LIN {X 0,Y 587.637,Z 719.821,A -85,B 0,C 180,E1 26964.756,E2 26964.756} C_VEL
LIN {X 0,Y 588.575,Z 722.928,A -85,B 0,C 180,E1 26962.657,E2 26962.657} C_VEL
LIN {X 0,Y 589.247,Z 724.472,A -85,B 0,C 180,E1 26961.936,E2 26961.936} C_VEL
LIN {X 0,Y 590.735,Z 728.438,A -85,B 0,C 180,E1 26960.6,E2 26960.6} C_VEL
LIN {X 0,Y 592.603,Z 733.926,A -85,B 0,C 180,E1 26959.233,E2 26959.233} C_VEL
LIN {X 0,Y 593.872,Z 738.208,A -85,B 0,C 180,E1 26958.376,E2 26958.376} C_VEL
LIN {X 0,Y 585.951,Z 770.314,A -85,B 0,C 180,E1 26955.875,E2 26955.875} C_VEL
LIN {X 0,Y 580.418,Z 801.749,A -85,B 0,C 180,E1 26953.509,E2 26953.509} C_VEL
LIN {X 0,Y 578.896,Z 823.206,A -85,B 0,C 180,E1 26951.811,E2 26951.811} C_VEL
LIN {X 0,Y 579.57,Z 841.188,A -85,B 0,C 180,E1 26950.31,E2 26950.31} C_VEL
LIN {X 0,Y 582.431,Z 858.387,A -85,B 0,C 180,E1 26948.793,E2 26948.793} C_VEL
LIN {X 0,Y 587.132,Z 873.472,A -85,B 0,C 180,E1 26947.396,E2 26947.396} C_VEL
LIN {X 0,Y 593.648,Z 887.403,A -85,B 0,C 180,E1 26946.053,E2 26946.053} C_VEL
LIN {X 0,Y 602.264,Z 900.569,A -85,B 0,C 180,E1 26944.733,E2 26944.733} C_VEL
LIN {X 0,Y 611.989,Z 911.844,A -85,B 0,C 180,E1 26943.565,E2 26943.565} C_VEL
LIN {X 0,Y 613.681,Z 913.685,A -85,B 0,C 180,E1 26943.378,E2 26943.378} C_VEL
LIN {X 0,Y 600.72,Z 934.889,A -85,B 0,C 180,E1 26942.747,E2 26942.747} C_VEL
LIN {X 0,Y 591.048,Z 953.679,A -85,B 0,C 180,E1 26942.084,E2 26942.084} C_VEL
LIN {X 0,Y 583.725,Z 969.894,A -85,B 0,C 180,E1 26941.455,E2 26941.455} C_VEL
LIN {X 0,Y 576.421,Z 987.193,A -85,B 0,C 180,E1 26940.746,E2 26940.746} C_VEL
LIN {X 0,Y 572.039,Z 1000.302,A -85,B 0,C 180,E1 26940.18,E2 26940.18} C_VEL
LIN {X 0,Y 569.588,Z 1022.689,A -85,B 0,C 180,E1 26939.955,E2 26939.955} C_VEL
LIN {X 0,Y 568.415,Z 1062.738,A -85,B 0,C 180,E1 26939.349,E2 26939.349} C_VEL
LIN {X 0,Y 567.38,Z 1084.854,A -85,B 0,C 180,E1 26938.837,E2 26938.837} C_VEL
LIN {X 0,Y 566.128,Z 1105.829,A -85,B 0,C 180,E1 26938.174,E2 26938.174} C_VEL
LIN {X 0,Y 564.559,Z 1128.324,A -85,B 0,C 180,E1 26937.264,E2 26937.264} C_VEL
LIN {X 0,Y 562.987,Z 1148.678,A -85,B 0,C 180,E1 26936.245,E2 26936.245} C_VEL
LIN {X 0,Y 561.314,Z 1168.753,A -85,B 0,C 180,E1 26935.026,E2 26935.026} C_VEL
LIN {X 0,Y 559.661,Z 1187.098,A -85,B 0,C 180,E1 26933.7,E2 26933.7} C_VEL
LIN {X 0,Y 558.095,Z 1204.72,A -85,B 0,C 180,E1 26932.21,E2 26932.21} C_VEL
LIN {X 0,Y 556.649,Z 1220.957,A -85,B 0,C 180,E1 26930.612,E2 26930.612} C_VEL
LIN {X 0,Y 555.379,Z 1235.689,A -85,B 0,C 180,E1 26928.907,E2 26928.907} C_VEL
LIN {X 0,Y 554.298,Z 1249.482,A -85,B 0,C 180,E1 26927.047,E2 26927.047} C_VEL
LIN {X 0,Y 553.424,Z 1261.927,A -85,B 0,C 180,E1 26925.078,E2 26925.078} C_VEL
LIN {X 0,Y 552.819,Z 1272.613,A -85,B 0,C 180,E1 26923.065,E2 26923.065} C_VEL
LIN {X 0,Y 552.412,Z 1281.385,A -85,B 0,C 180,E1 26921.06,E2 26921.06} C_VEL
LIN {X 0,Y 552.19,Z 1288.893,A -85,B 0,C 180,E1 26918.957,E2 26918.957} C_VEL
LIN {X 0,Y 552.095,Z 1294.66,A -85,B 0,C 180,E1 26916.864,E2 26916.864} C_VEL
LIN {X 0,Y 552.078,Z 1298.97,A -85,B 0,C 180,E1 26914.673,E2 26914.673} C_VEL
LIN {X 0,Y 552.098,Z 1301.66,A -85,B 0,C 180,E1 26912.49,E2 26912.49} C_VEL
LIN {X 0,Y 552.111,Z 1302.611,A -85,B 0,C 180,E1 26910.414,E2 26910.414} C_VEL
LIN {X 0,Y 552.119,Z 1302.041,A -85,B 0,C 180,E1 26908.234,E2 26908.234} C_VEL
LIN {X 0,Y 552.092,Z 1299.995,A -85,B 0,C 180,E1 26906.156,E2 26906.156} C_VEL
LIN {X 0,Y 552.096,Z 1296.342,A -85,B 0,C 180,E1 26904.073,E2 26904.073} C_VEL
LIN {X 0,Y 552.146,Z 1291.188,A -85,B 0,C 180,E1 26901.983,E2 26901.983} C_VEL
LIN {X 0,Y 552.298,Z 1284.244,A -85,B 0,C 180,E1 26899.885,E2 26899.885} C_VEL
LIN {X 0,Y 552.609,Z 1275.501,A -85,B 0,C 180,E1 26897.777,E2 26897.777} C_VEL
LIN {X 0,Y 553.09,Z 1265.374,A -85,B 0,C 180,E1 26895.766,E2 26895.766} C_VEL
LIN {X 0,Y 553.776,Z 1253.837,A -85,B 0,C 180,E1 26893.854,E2 26893.854} C_VEL
LIN {X 0,Y 554.714,Z 1240.173,A -85,B 0,C 180,E1 26891.937,E2 26891.937} C_VEL
LIN {X 0,Y 555.856,Z 1225.016,A -85,B 0,C 180,E1 26890.123,E2 26890.123} C_VEL
LIN {X 0,Y 557.166,Z 1208.907,A -85,B 0,C 180,E1 26888.47,E2 26888.47} C_VEL
LIN {X 0,Y 558.616,Z 1191.119,A -85,B 0,C 180,E1 26886.92,E2 26886.92} C_VEL
LIN {X 0,Y 560.211,Z 1171.724,A -85,B 0,C 180,E1 26885.481,E2 26885.481} C_VEL
LIN {X 0,Y 561.815,Z 1151.511,A -85,B 0,C 180,E1 26884.21,E2 26884.21} C_VEL
LIN {X 0,Y 563.458,Z 1130.214,A -85,B 0,C 180,E1 26883.094,E2 26883.094} C_VEL
LIN {X 0,Y 565.016,Z 1107.978,A -85,B 0,C 180,E1 26882.147,E2 26882.147} C_VEL
LIN {X 0,Y 566.431,Z 1085.264,A -85,B 0,C 180,E1 26881.387,E2 26881.387} C_VEL
LIN {X 0,Y 567.595,Z 1062.247,A -85,B 0,C 180,E1 26880.821,E2 26880.821} C_VEL
LIN {X 0,Y 568.909,Z 1024.211,A -85,B 0,C 180,E1 26880.177,E2 26880.177} C_VEL
LIN {X 0,Y 570.051,Z 1012.277,A -85,B 0,C 180,E1 26880.006,E2 26880.006} C_VEL
LIN {X 0,Y 578.286,Z 988.02,A -85,B 0,C 180,E1 26878.869,E2 26878.869} C_VEL
LIN {X 0,Y 585.721,Z 971.102,A -85,B 0,C 180,E1 26878.163,E2 26878.163} C_VEL
LIN {X 0,Y 597.338,Z 946.651,A -85,B 0,C 180,E1 26877.213,E2 26877.213} C_VEL
LIN {X 0,Y 608.71,Z 926.849,A -85,B 0,C 180,E1 26876.56,E2 26876.56} C_VEL
LIN {X 0,Y 615.537,Z 915.878,A -85,B 0,C 180,E1 26876.237,E2 26876.237} C_VEL
LIN {X 0,Y 605.204,Z 904.179,A -85,B 0,C 180,E1 26875.032,E2 26875.032} C_VEL
LIN {X 0,Y 596.035,Z 890.457,A -85,B 0,C 180,E1 26873.714,E2 26873.714} C_VEL
LIN {X 0,Y 588.846,Z 875.63,A -85,B 0,C 180,E1 26872.386,E2 26872.386} C_VEL
LIN {X 0,Y 583.433,Z 859.428,A -85,B 0,C 180,E1 26871.025,E2 26871.025} C_VEL
LIN {X 0,Y 579.733,Z 840.872,A -85,B 0,C 180,E1 26869.57,E2 26869.57} C_VEL
LIN {X 0,Y 578.123,Z 820.933,A -85,B 0,C 180,E1 26868.117,E2 26868.117} C_VEL
LIN {X 0,Y 578.452,Z 797.639,A -85,B 0,C 180,E1 26866.53,E2 26866.53} C_VEL
LIN {X 0,Y 583.409,Z 741.175,A -85,B 0,C 180,E1 26862.876,E2 26862.876} C_VEL
LIN {X 0,Y 584.291,Z 731.836,A -85,B 0,C 180,E1 26862.263,E2 26862.263} C_VEL
LIN {X 0,Y 572.986,Z 706.025,A -85,B 0,C 180,E1 26859.37,E2 26859.37} C_VEL
LIN {X 0,Y 570.213,Z 699.791,A -85,B 0,C 180,E1 26858.62,E2 26858.62} C_VEL
LIN {X 0,Y 572.694,Z 699.884,A -85,B 0,C 180,E1 26858.135,E2 26858.135} C_VEL
LIN {X 0,Y 575.711,Z 710.211,A -85,B 0,C 180,E1 26856.44,E2 26856.44} C_VEL
LIN {X 0,Y 576.967,Z 715.049,A -85,B 0,C 180,E1 26855.777,E2 26855.777} C_VEL
LIN {X 0,Y 580.175,Z 722.589,A -85,B 0,C 180,E1 26855.137,E2 26855.137} C_VEL
LIN {X 0,Y 582.997,Z 739.875,A -85,B 0,C 180,E1 26854.313,E2 26854.313} C_VEL
LIN {X 0,Y 576.786,Z 834.739,A -85,B 0,C 180,E1 26852.485,E2 26852.485} C_VEL
LIN {X 0,Y 572.384,Z 927.388,A -85,B 0,C 180,E1 26850.83,E2 26850.83} C_VEL
LIN {X 0,Y 569.328,Z 1016.488,A -85,B 0,C 180,E1 26849.344,E2 26849.344} C_VEL
LIN {X 0,Y 568.303,Z 1039.379,A -85,B 0,C 180,E1 26848.764,E2 26848.764} C_VEL
LIN {X 0,Y 567.075,Z 1060.726,A -85,B 0,C 180,E1 26848.046,E2 26848.046} C_VEL
LIN {X 0,Y 565.582,Z 1082.832,A -85,B 0,C 180,E1 26847.104,E2 26847.104} C_VEL
LIN {X 0,Y 564.08,Z 1102.487,A -85,B 0,C 180,E1 26846.079,E2 26846.079} C_VEL
LIN {X 0,Y 562.432,Z 1121.912,A -85,B 0,C 180,E1 26844.863,E2 26844.863} C_VEL
LIN {X 0,Y 560.743,Z 1140.326,A -85,B 0,C 180,E1 26843.487,E2 26843.487} C_VEL
LIN {X 0,Y 559.062,Z 1157.806,A -85,B 0,C 180,E1 26841.95,E2 26841.95} C_VEL
LIN {X 0,Y 557.574,Z 1173.309,A -85,B 0,C 180,E1 26840.359,E2 26840.359} C_VEL
LIN {X 0,Y 556.152,Z 1188.302,A -85,B 0,C 180,E1 26838.556,E2 26838.556} C_VEL
LIN {X 0,Y 554.91,Z 1201.645,A -85,B 0,C 180,E1 26836.649,E2 26836.649} C_VEL
LIN {X 0,Y 553.906,Z 1213.516,A -85,B 0,C 180,E1 26834.639,E2 26834.639} C_VEL
LIN {X 0,Y 553.135,Z 1223.889,A -85,B 0,C 180,E1 26832.528,E2 26832.528} C_VEL
LIN {X 0,Y 552.629,Z 1232.359,A -85,B 0,C 180,E1 26830.424,E2 26830.424} C_VEL
LIN {X 0,Y 552.285,Z 1239.262,A -85,B 0,C 180,E1 26828.223,E2 26828.223} C_VEL
LIN {X 0,Y 552.102,Z 1244.436,A -85,B 0,C 180,E1 26826.03,E2 26826.03} C_VEL
LIN {X 0,Y 552.013,Z 1248.008,A -85,B 0,C 180,E1 26823.843,E2 26823.843} C_VEL
LIN {X 0,Y 551.984,Z 1249.897,A -85,B 0,C 180,E1 26821.661,E2 26821.661} C_VEL
LIN {X 0,Y 551.985,Z 1250.235,A -85,B 0,C 180,E1 26819.377,E2 26819.377} C_VEL
LIN {X 0,Y 551.983,Z 1248.966,A -85,B 0,C 180,E1 26817.136,E2 26817.136} C_VEL
LIN {X 0,Y 552.025,Z 1246.172,A -85,B 0,C 180,E1 26815.012,E2 26815.012} C_VEL
LIN {X 0,Y 552.147,Z 1241.721,A -85,B 0,C 180,E1 26812.822,E2 26812.822} C_VEL
LIN {X 0,Y 552.383,Z 1235.625,A -85,B 0,C 180,E1 26810.624,E2 26810.624} C_VEL
LIN {X 0,Y 552.774,Z 1228.041,A -85,B 0,C 180,E1 26808.523,E2 26808.523} C_VEL
LIN {X 0,Y 553.376,Z 1218.633,A -85,B 0,C 180,E1 26806.414,E2 26806.414} C_VEL
LIN {X 0,Y 554.213,Z 1207.87,A -85,B 0,C 180,E1 26804.406,E2 26804.406} C_VEL
LIN {X 0,Y 555.271,Z 1195.735,A -85,B 0,C 180,E1 26802.499,E2 26802.499} C_VEL
LIN {X 0,Y 556.51,Z 1182.18,A -85,B 0,C 180,E1 26800.695,E2 26800.695} C_VEL
LIN {X 0,Y 558.041,Z 1166.325,A -85,B 0,C 180,E1 26798.891,E2 26798.891} C_VEL
LIN {X 0,Y 559.663,Z 1149.96,A -85,B 0,C 180,E1 26797.3,E2 26797.3} C_VEL
LIN {X 0,Y 561.374,Z 1132.001,A -85,B 0,C 180,E1 26795.816,E2 26795.816} C_VEL
LIN {X 0,Y 563.033,Z 1113.854,A -85,B 0,C 180,E1 26794.547,E2 26794.547} C_VEL
LIN {X 0,Y 564.757,Z 1093.28,A -85,B 0,C 180,E1 26793.332,E2 26793.332} C_VEL
LIN {X 0,Y 566.359,Z 1072.777,A -85,B 0,C 180,E1 26792.334,E2 26792.334} C_VEL
LIN {X 0,Y 567.755,Z 1051.302,A -85,B 0,C 180,E1 26791.493,E2 26791.493} C_VEL
LIN {X 0,Y 568.91,Z 1029.578,A -85,B 0,C 180,E1 26790.838,E2 26790.838} C_VEL
LIN {X 0,Y 569.869,Z 1006.211,A -85,B 0,C 180,E1 26790.329,E2 26790.329} C_VEL
LIN {X 0,Y 576.672,Z 748.494,A -85,B 0,C 180,E1 26786.536,E2 26786.536} C_VEL
LIN {X 0,Y 576.781,Z 737.467,A -85,B 0,C 180,E1 26786.358,E2 26786.358} C_VEL
LIN {X 0,Y 571.105,Z 712.252,A -85,B 0,C 180,E1 26785.574,E2 26785.574} C_VEL
LIN {X 0,Y 567.095,Z 704.126,A -85,B 0,C 180,E1 26785.161,E2 26785.161} C_VEL
LIN {X 0,Y 560.021,Z 682.503,A -85,B 0,C 180,E1 26782.611,E2 26782.611} C_VEL
LIN {X 0,Y 553.503,Z 663.719,A -85,B 0,C 180,E1 26780.315,E2 26780.315} C_VEL
LIN {X 0,Y 553.497,Z 663.72,A -85,B 0,C 180,E1 26776.932,E2 26776.932} C_VEL
LIN {X 0,Y 553.509,Z 663.725,A -85,B 0,C 180,E1 26773.494,E2 26773.494} C_VEL
LIN {X 0,Y 553.506,Z 663.721,A -85,B 0,C 180,E1 26770.565,E2 26770.565} C_VEL
LIN {X 0,Y 552.506,Z 663.847,A -85,B 0,C 180,E1 26769.768,E2 26769.768} C_VEL
LIN {X 0,Y 546.084,Z 664.643,A -85,B 0,C 180,E1 26767.529,E2 26767.529} C_VEL
LIN {X 0,Y 545.549,Z 664.706,A -85,B 0,C 180,E1 26766.946,E2 26766.946} C_VEL
LIN {X 0,Y 545.555,Z 664.708,A -85,B 0,C 180,E1 26763.609,E2 26763.609} C_VEL
LIN {X 0,Y 545.566,Z 664.706,A -85,B 0,C 180,E1 26760.11,E2 26760.11} C_VEL
LIN {X 0,Y 545.553,Z 664.71,A -85,B 0,C 180,E1 26756.683,E2 26756.683} C_VEL
LIN {X 0,Y 545.565,Z 664.712,A -85,B 0,C 180,E1 26753.322,E2 26753.322} C_VEL
LIN {X 0,Y 545.567,Z 664.709,A -85,B 0,C 180,E1 26749.821,E2 26749.821} C_VEL
LIN {X 0,Y 545.555,Z 664.713,A -85,B 0,C 180,E1 26746.396,E2 26746.396} C_VEL
LIN {X 0,Y 545.559,Z 664.703,A -85,B 0,C 180,E1 26743.03,E2 26743.03} C_VEL
LIN {X 0,Y 545.552,Z 664.712,A -85,B 0,C 180,E1 26739.709,E2 26739.709} C_VEL
LIN {X 0,Y 545.565,Z 664.709,A -85,B 0,C 180,E1 26736.315,E2 26736.315} C_VEL
LIN {X 0,Y 545.552,Z 664.707,A -85,B 0,C 180,E1 26732.838,E2 26732.838} C_VEL
LIN {X 0,Y 545.548,Z 664.703,A -85,B 0,C 180,E1 26729.476,E2 26729.476} C_VEL
LIN {X 0,Y 545.553,Z 664.702,A -85,B 0,C 180,E1 26726.113,E2 26726.113} C_VEL
LIN {X 0,Y 545.562,Z 664.702,A -85,B 0,C 180,E1 26722.631,E2 26722.631} C_VEL
LIN {X 0,Y 545.549,Z 664.704,A -85,B 0,C 180,E1 26719.227,E2 26719.227} C_VEL
LIN {X 0,Y 545.561,Z 664.706,A -85,B 0,C 180,E1 26715.893,E2 26715.893} C_VEL
LIN {X 0,Y 545.567,Z 664.709,A -85,B 0,C 180,E1 26712.51,E2 26712.51} C_VEL
LIN {X 0,Y 545.561,Z 664.712,A -85,B 0,C 180,E1 26709.062,E2 26709.062} C_VEL
LIN {X 0,Y 545.562,Z 664.713,A -85,B 0,C 180,E1 26705.648,E2 26705.648} C_VEL
LIN {X 0,Y 545.556,Z 664.709,A -85,B 0,C 180,E1 26702.258,E2 26702.258} C_VEL
LIN {X 0,Y 545.565,Z 664.71,A -85,B 0,C 180,E1 26698.86,E2 26698.86} C_VEL
LIN {X 0,Y 545.554,Z 664.716,A -85,B 0,C 180,E1 26695.379,E2 26695.379} C_VEL
LIN {X 0,Y 545.551,Z 664.714,A -85,B 0,C 180,E1 26691.991,E2 26691.991} C_VEL
LIN {X 0,Y 545.587,Z 664.857,A -85,B 0,C 180,E1 26689.554,E2 26689.554} C_VEL
LIN {X 0,Y 554.863,Z 689.261,A -85,B 0,C 180,E1 26686.501,E2 26686.501} C_VEL
LIN {X 0,Y 562.764,Z 711.514,A -85,B 0,C 180,E1 26683.91,E2 26683.91} C_VEL
LIN {X 0,Y 565.161,Z 719.188,A -85,B 0,C 180,E1 26683.059,E2 26683.059} C_VEL
LIN {X 0,Y 562.422,Z 755.919,A -85,B 0,C 180,E1 26680.059,E2 26680.059} C_VEL
LIN {X 0,Y 559.159,Z 801.286,A -85,B 0,C 180,E1 26676.419,E2 26676.419} C_VEL
LIN {X 0,Y 556.143,Z 848.128,A -85,B 0,C 180,E1 26672.714,E2 26672.714} C_VEL
LIN {X 0,Y 553.504,Z 895.199,A -85,B 0,C 180,E1 26669.038,E2 26669.038} C_VEL
LIN {X 0,Y 553.065,Z 904.913,A -85,B 0,C 180,E1 26668.313,E2 26668.313} C_VEL
LIN {X 0,Y 553.968,Z 914.616,A -85,B 0,C 180,E1 26668.102,E2 26668.102} C_VEL
LIN {X 0,Y 550.539,Z 1049.576,A -85,B 0,C 180,E1 26665.712,E2 26665.712} C_VEL
LIN {X 0,Y 550.165,Z 1066.208,A -85,B 0,C 180,E1 26665.226,E2 26665.226} C_VEL
LIN {X 0,Y 549.614,Z 1082.443,A -85,B 0,C 180,E1 26664.551,E2 26664.551} C_VEL
LIN {X 0,Y 548.912,Z 1098.012,A -85,B 0,C 180,E1 26663.682,E2 26663.682} C_VEL
LIN {X 0,Y 548.208,Z 1111.947,A -85,B 0,C 180,E1 26662.691,E2 26662.691} C_VEL
LIN {X 0,Y 547.447,Z 1125.469,A -85,B 0,C 180,E1 26661.482,E2 26661.482} C_VEL
LIN {X 0,Y 546.781,Z 1136.869,A -85,B 0,C 180,E1 26660.22,E2 26660.22} C_VEL
LIN {X 0,Y 546.158,Z 1147.204,A -85,B 0,C 180,E1 26658.797,E2 26658.797} C_VEL
LIN {X 0,Y 545.662,Z 1156.069,A -85,B 0,C 180,E1 26657.269,E2 26657.269} C_VEL
LIN {X 0,Y 545.289,Z 1163.329,A -85,B 0,C 180,E1 26655.638,E2 26655.638} C_VEL
LIN {X 0,Y 545.071,Z 1168.797,A -85,B 0,C 180,E1 26653.983,E2 26653.983} C_VEL
LIN {X 0,Y 544.954,Z 1172.679,A -85,B 0,C 180,E1 26652.181,E2 26652.181} C_VEL
LIN {X 0,Y 544.948,Z 1174.629,A -85,B 0,C 180,E1 26650.445,E2 26650.445} C_VEL
LIN {X 0,Y 545.045,Z 1174.714,A -85,B 0,C 180,E1 26648.599,E2 26648.599} C_VEL
LIN {X 0,Y 545.221,Z 1173.143,A -85,B 0,C 180,E1 26646.952,E2 26646.952} C_VEL
LIN {X 0,Y 545.552,Z 1169.515,A -85,B 0,C 180,E1 26645.153,E2 26645.153} C_VEL
LIN {X 0,Y 546.033,Z 1164.264,A -85,B 0,C 180,E1 26643.464,E2 26643.464} C_VEL
LIN {X 0,Y 546.699,Z 1157.01,A -85,B 0,C 180,E1 26641.782,E2 26641.782} C_VEL
LIN {X 0,Y 547.478,Z 1148.769,A -85,B 0,C 180,E1 26640.314,E2 26640.314} C_VEL
LIN {X 0,Y 548.442,Z 1138.381,A -85,B 0,C 180,E1 26638.851,E2 26638.851} C_VEL
LIN {X 0,Y 549.401,Z 1127.311,A -85,B 0,C 180,E1 26637.601,E2 26637.601} C_VEL
LIN {X 0,Y 550.437,Z 1114.18,A -85,B 0,C 180,E1 26636.407,E2 26636.407} C_VEL
LIN {X 0,Y 551.384,Z 1100.664,A -85,B 0,C 180,E1 26635.423,E2 26635.423} C_VEL
LIN {X 0,Y 552.318,Z 1085.265,A -85,B 0,C 180,E1 26634.546,E2 26634.546} C_VEL
LIN {X 0,Y 552.969,Z 1070.158,A -85,B 0,C 180,E1 26633.902,E2 26633.902} C_VEL
LIN {X 0,Y 553.451,Z 1053.734,A -85,B 0,C 180,E1 26633.399,E2 26633.399} C_VEL
LIN {X 0,Y 556.81,Z 986.578,A -85,B 0,C 180,E1 26631.834,E2 26631.834} C_VEL
LIN {X 0,Y 560.911,Z 918.315,A -85,B 0,C 180,E1 26630.302,E2 26630.302} C_VEL
LIN {X 0,Y 566.056,Z 873.39,A -85,B 0,C 180,E1 26626.412,E2 26626.412} C_VEL
LIN {X 0,Y 571.814,Z 833.12,A -85,B 0,C 180,E1 26622.811,E2 26622.811} C_VEL
LIN {X 0,Y 578.862,Z 793.757,A -85,B 0,C 180,E1 26619.155,E2 26619.155} C_VEL
LIN {X 0,Y 585.523,Z 763.603,A -85,B 0,C 180,E1 26616.233,E2 26616.233} C_VEL
LIN {X 0,Y 588.504,Z 750.811,A -85,B 0,C 180,E1 26614.897,E2 26614.897} C_VEL
LIN {X 0,Y 586.346,Z 742.225,A -85,B 0,C 180,E1 26613.024,E2 26613.024} C_VEL
LIN {X 0,Y 584.554,Z 735.363,A -85,B 0,C 180,E1 26611.134,E2 26611.134} C_VEL
LIN {X 0,Y 583.377,Z 731.221,A -85,B 0,C 180,E1 26609.552,E2 26609.552} C_VEL
LIN {X 0,Y 582.906,Z 728.956,A -85,B 0,C 180,E1 26608.454,E2 26608.454} C_VEL
LIN {X 0,Y 582.719,Z 726.445,A -85,B 0,C 180,E1 26606.223,E2 26606.223} C_VEL
LIN {X 0,Y 583.098,Z 726.497,A -85,B 0,C 180,E1 26604.698,E2 26604.698} C_VEL
LIN {X 0,Y 584.121,Z 729.672,A -85,B 0,C 180,E1 26602.578,E2 26602.578} C_VEL
LIN {X 0,Y 585.59,Z 733.498,A -85,B 0,C 180,E1 26601.071,E2 26601.071} C_VEL
LIN {X 0,Y 587.4,Z 739.28,A -85,B 0,C 180,E1 26599.54,E2 26599.54} C_VEL
LIN {X 0,Y 588.338,Z 743.262,A -85,B 0,C 180,E1 26598.745,E2 26598.745} C_VEL
LIN {X 0,Y 580.343,Z 773.332,A -85,B 0,C 180,E1 26596.352,E2 26596.352} C_VEL
LIN {X 0,Y 574.439,Z 804.082,A -85,B 0,C 180,E1 26593.986,E2 26593.986} C_VEL
LIN {X 0,Y 572.592,Z 825.779,A -85,B 0,C 180,E1 26592.233,E2 26592.233} C_VEL
LIN {X 0,Y 573.004,Z 843.762,A -85,B 0,C 180,E1 26590.701,E2 26590.701} C_VEL
LIN {X 0,Y 575.6,Z 861.112,A -85,B 0,C 180,E1 26589.138,E2 26589.138} C_VEL
LIN {X 0,Y 580.048,Z 876.32,A -85,B 0,C 180,E1 26587.699,E2 26587.699} C_VEL
LIN {X 0,Y 586.616,Z 890.959,A -85,B 0,C 180,E1 26586.259,E2 26586.259} C_VEL
LIN {X 0,Y 595.004,Z 904.185,A -85,B 0,C 180,E1 26584.907,E2 26584.907} C_VEL
LIN {X 0,Y 604.548,Z 916.003,A -85,B 0,C 180,E1 26583.682,E2 26583.682} C_VEL
LIN {X 0,Y 592.21,Z 936.838,A -85,B 0,C 180,E1 26583.047,E2 26583.047} C_VEL
LIN {X 0,Y 582.805,Z 955.77,A -85,B 0,C 180,E1 26582.361,E2 26582.361} C_VEL
LIN {X 0,Y 576.479,Z 969.641,A -85,B 0,C 180,E1 26581.82,E2 26581.82} C_VEL
LIN {X 0,Y 569.168,Z 987.099,A -85,B 0,C 180,E1 26581.095,E2 26581.095} C_VEL
LIN {X 0,Y 564.903,Z 999.752,A -85,B 0,C 180,E1 26580.541,E2 26580.541} C_VEL
LIN {X 0,Y 562.392,Z 1022.537,A -85,B 0,C 180,E1 26580.308,E2 26580.308} C_VEL
LIN {X 0,Y 561.125,Z 1062.761,A -85,B 0,C 180,E1 26579.685,E2 26579.685} C_VEL
LIN {X 0,Y 560.025,Z 1085.237,A -85,B 0,C 180,E1 26579.155,E2 26579.155} C_VEL
LIN {X 0,Y 558.673,Z 1106.781,A -85,B 0,C 180,E1 26578.457,E2 26578.457} C_VEL
LIN {X 0,Y 557.118,Z 1128.02,A -85,B 0,C 180,E1 26577.582,E2 26577.582} C_VEL
LIN {X 0,Y 555.463,Z 1148.633,A -85,B 0,C 180,E1 26576.536,E2 26576.536} C_VEL
LIN {X 0,Y 553.759,Z 1168.215,A -85,B 0,C 180,E1 26575.335,E2 26575.335} C_VEL
LIN {X 0,Y 552.06,Z 1186.412,A -85,B 0,C 180,E1 26574.007,E2 26574.007} C_VEL
LIN {X 0,Y 550.337,Z 1204.84,A -85,B 0,C 180,E1 26572.427,E2 26572.427} C_VEL
LIN {X 0,Y 548.832,Z 1221.013,A -85,B 0,C 180,E1 26570.808,E2 26570.808} C_VEL
LIN {X 0,Y 547.436,Z 1236.626,A -85,B 0,C 180,E1 26568.971,E2 26568.971} C_VEL
LIN {X 0,Y 546.353,Z 1249.898,A -85,B 0,C 180,E1 26567.135,E2 26567.135} C_VEL
LIN {X 0,Y 545.43,Z 1262.506,A -85,B 0,C 180,E1 26565.087,E2 26565.087} C_VEL
LIN {X 0,Y 544.818,Z 1273.091,A -85,B 0,C 180,E1 26563.045,E2 26563.045} C_VEL
LIN {X 0,Y 544.404,Z 1281.713,A -85,B 0,C 180,E1 26561.01,E2 26561.01} C_VEL
LIN {X 0,Y 544.181,Z 1289.378,A -85,B 0,C 180,E1 26558.771,E2 26558.771} C_VEL
LIN {X 0,Y 544.09,Z 1295.005,A -85,B 0,C 180,E1 26556.647,E2 26556.647} C_VEL
LIN {X 0,Y 544.089,Z 1298.9,A -85,B 0,C 180,E1 26554.531,E2 26554.531} C_VEL
LIN {X 0,Y 544.107,Z 1301.483,A -85,B 0,C 180,E1 26552.21,E2 26552.21} C_VEL
LIN {X 0,Y 544.13,Z 1302.29,A -85,B 0,C 180,E1 26550.104,E2 26550.104} C_VEL
LIN {X 0,Y 544.122,Z 1301.506,A -85,B 0,C 180,E1 26547.998,E2 26547.998} C_VEL
LIN {X 0,Y 544.098,Z 1299.314,A -85,B 0,C 180,E1 26545.889,E2 26545.889} C_VEL
LIN {X 0,Y 544.107,Z 1295.467,A -85,B 0,C 180,E1 26543.774,E2 26543.774} C_VEL
LIN {X 0,Y 544.174,Z 1289.758,A -85,B 0,C 180,E1 26541.546,E2 26541.546} C_VEL
LIN {X 0,Y 544.339,Z 1282.608,A -85,B 0,C 180,E1 26539.414,E2 26539.414} C_VEL
LIN {X 0,Y 544.715,Z 1273.486,A -85,B 0,C 180,E1 26537.274,E2 26537.274} C_VEL
LIN {X 0,Y 545.264,Z 1262.948,A -85,B 0,C 180,E1 26535.231,E2 26535.231} C_VEL
LIN {X 0,Y 546.05,Z 1250.992,A -85,B 0,C 180,E1 26533.273,E2 26533.273} C_VEL
LIN {X 0,Y 547.078,Z 1237.005,A -85,B 0,C 180,E1 26531.345,E2 26531.345} C_VEL
LIN {X 0,Y 548.304,Z 1221.781,A -85,B 0,C 180,E1 26529.559,E2 26529.559} C_VEL
LIN {X 0,Y 549.8,Z 1204.552,A -85,B 0,C 180,E1 26527.828,E2 26527.828} C_VEL
LIN {X 0,Y 551.31,Z 1187.216,A -85,B 0,C 180,E1 26526.335,E2 26526.335} C_VEL
LIN {X 0,Y 553.009,Z 1167.711,A -85,B 0,C 180,E1 26524.912,E2 26524.912} C_VEL
LIN {X 0,Y 554.595,Z 1148.502,A -85,B 0,C 180,E1 26523.728,E2 26523.728} C_VEL
LIN {X 0,Y 556.329,Z 1126.757,A -85,B 0,C 180,E1 26522.605,E2 26522.605} C_VEL
LIN {X 0,Y 557.962,Z 1104.6,A -85,B 0,C 180,E1 26521.676,E2 26521.676} C_VEL
LIN {X 0,Y 559.476,Z 1081.506,A -85,B 0,C 180,E1 26520.913,E2 26520.913} C_VEL
LIN {X 0,Y 560.794,Z 1057.496,A -85,B 0,C 180,E1 26520.333,E2 26520.333} C_VEL
LIN {X 0,Y 562.329,Z 1020.095,A -85,B 0,C 180,E1 26519.709,E2 26519.709} C_VEL
LIN {X 0,Y 563.455,Z 1009.36,A -85,B 0,C 180,E1 26519.559,E2 26519.559} C_VEL
LIN {X 0,Y 572.631,Z 983.532,A -85,B 0,C 180,E1 26518.35,E2 26518.35} C_VEL
LIN {X 0,Y 580.823,Z 965.891,A -85,B 0,C 180,E1 26517.629,E2 26517.629} C_VEL
LIN {X 0,Y 589.845,Z 946.692,A -85,B 0,C 180,E1 26516.869,E2 26516.869} C_VEL
LIN {X 0,Y 601.196,Z 926.722,A -85,B 0,C 180,E1 26516.197,E2 26516.197} C_VEL
LIN {X 0,Y 606.49,Z 918.028,A -85,B 0,C 180,E1 26515.929,E2 26515.929} C_VEL
LIN {X 0,Y 596.592,Z 905.997,A -85,B 0,C 180,E1 26514.708,E2 26514.708} C_VEL
LIN {X 0,Y 587.93,Z 892.207,A -85,B 0,C 180,E1 26513.392,E2 26513.392} C_VEL
LIN {X 0,Y 580.965,Z 876.905,A -85,B 0,C 180,E1 26512.023,E2 26512.023} C_VEL
LIN {X 0,Y 575.96,Z 860.908,A -85,B 0,C 180,E1 26510.679,E2 26510.679} C_VEL
LIN {X 0,Y 572.512,Z 842.361,A -85,B 0,C 180,E1 26509.217,E2 26509.217} C_VEL
LIN {X 0,Y 571.062,Z 821.442,A -85,B 0,C 180,E1 26507.682,E2 26507.682} C_VEL
LIN {X 0,Y 571.641,Z 797.908,A -85,B 0,C 180,E1 26506.068,E2 26506.068} C_VEL
LIN {X 0,Y 576.658,Z 743.739,A -85,B 0,C 180,E1 26502.529,E2 26502.529} C_VEL
LIN {X 0,Y 577.396,Z 735.075,A -85,B 0,C 180,E1 26501.947,E2 26501.947} C_VEL
LIN {X 0,Y 565.979,Z 708.93,A -85,B 0,C 180,E1 26498.971,E2 26498.971} C_VEL
LIN {X 0,Y 565.168,Z 707.036,A -85,B 0,C 180,E1 26498.719,E2 26498.719} C_VEL
LIN {X 0,Y 568.008,Z 706.852,A -85,B 0,C 180,E1 26498.162,E2 26498.162} C_VEL
LIN {X 0,Y 570.477,Z 715.922,A -85,B 0,C 180,E1 26496.652,E2 26496.652} C_VEL
LIN {X 0,Y 575.181,Z 726.389,A -85,B 0,C 180,E1 26495.63,E2 26495.63} C_VEL
LIN {X 0,Y 577.487,Z 742.124,A -85,B 0,C 180,E1 26494.854,E2 26494.854} C_VEL
LIN {X 0,Y 570.93,Z 831.791,A -85,B 0,C 180,E1 26493.069,E2 26493.069} C_VEL
LIN {X 0,Y 566.314,Z 916.888,A -85,B 0,C 180,E1 26491.482,E2 26491.482} C_VEL
LIN {X 0,Y 562.382,Z 1017.517,A -85,B 0,C 180,E1 26489.735,E2 26489.735} C_VEL
LIN {X 0,Y 561.272,Z 1040.63,A -85,B 0,C 180,E1 26489.133,E2 26489.133} C_VEL
LIN {X 0,Y 559.926,Z 1062.321,A -85,B 0,C 180,E1 26488.383,E2 26488.383} C_VEL
LIN {X 0,Y 558.398,Z 1083.529,A -85,B 0,C 180,E1 26487.458,E2 26487.458} C_VEL
LIN {X 0,Y 556.767,Z 1103.605,A -85,B 0,C 180,E1 26486.39,E2 26486.39} C_VEL
LIN {X 0,Y 555.04,Z 1122.919,A -85,B 0,C 180,E1 26485.16,E2 26485.16} C_VEL
LIN {X 0,Y 553.264,Z 1141.219,A -85,B 0,C 180,E1 26483.767,E2 26483.767} C_VEL
LIN {X 0,Y 551.493,Z 1158.616,A -85,B 0,C 180,E1 26482.211,E2 26482.211} C_VEL
LIN {X 0,Y 549.856,Z 1174.686,A -85,B 0,C 180,E1 26480.526,E2 26480.526} C_VEL
LIN {X 0,Y 548.384,Z 1189.406,A -85,B 0,C 180,E1 26478.718,E2 26478.718} C_VEL
LIN {X 0,Y 547.041,Z 1203.168,A -85,B 0,C 180,E1 26476.708,E2 26476.708} C_VEL
LIN {X 0,Y 546.024,Z 1214.427,A -85,B 0,C 180,E1 26474.746,E2 26474.746} C_VEL
LIN {X 0,Y 545.212,Z 1224.715,A -85,B 0,C 180,E1 26472.606,E2 26472.606} C_VEL
LIN {X 0,Y 544.677,Z 1233.106,A -85,B 0,C 180,E1 26470.471,E2 26470.471} C_VEL
LIN {X 0,Y 544.315,Z 1239.954,A -85,B 0,C 180,E1 26468.238,E2 26468.238} C_VEL
LIN {X 0,Y 544.119,Z 1245.034,A -85,B 0,C 180,E1 26466.013,E2 26466.013} C_VEL
LIN {X 0,Y 544.024,Z 1248.515,A -85,B 0,C 180,E1 26463.794,E2 26463.794} C_VEL
LIN {X 0,Y 543.993,Z 1250.355,A -85,B 0,C 180,E1 26461.58,E2 26461.58} C_VEL
LIN {X 0,Y 543.994,Z 1250.612,A -85,B 0,C 180,E1 26459.368,E2 26459.368} C_VEL
LIN {X 0,Y 543.994,Z 1249.367,A -85,B 0,C 180,E1 26457.139,E2 26457.139} C_VEL
LIN {X 0,Y 544.04,Z 1246.498,A -85,B 0,C 180,E1 26454.939,E2 26454.939} C_VEL
LIN {X 0,Y 544.17,Z 1241.999,A -85,B 0,C 180,E1 26452.716,E2 26452.716} C_VEL
LIN {X 0,Y 544.424,Z 1235.847,A -85,B 0,C 180,E1 26450.486,E2 26450.486} C_VEL
LIN {X 0,Y 544.845,Z 1228.218,A -85,B 0,C 180,E1 26448.354,E2 26448.354} C_VEL
LIN {X 0,Y 545.484,Z 1218.744,A -85,B 0,C 180,E1 26446.214,E2 26446.214} C_VEL
LIN {X 0,Y 546.371,Z 1207.896,A -85,B 0,C 180,E1 26444.176,E2 26444.176} C_VEL
LIN {X 0,Y 547.493,Z 1195.687,A -85,B 0,C 180,E1 26442.242,E2 26442.242} C_VEL
LIN {X 0,Y 548.834,Z 1181.694,A -85,B 0,C 180,E1 26440.374,E2 26440.374} C_VEL
LIN {X 0,Y 550.407,Z 1166.011,A -85,B 0,C 180,E1 26438.583,E2 26438.583} C_VEL
LIN {X 0,Y 552.101,Z 1149.506,A -85,B 0,C 180,E1 26436.971,E2 26436.971} C_VEL
LIN {X 0,Y 553.91,Z 1131.46,A -85,B 0,C 180,E1 26435.469,E2 26435.469} C_VEL
LIN {X 0,Y 555.633,Z 1113.098,A -85,B 0,C 180,E1 26434.183,E2 26434.183} C_VEL
LIN {X 0,Y 557.42,Z 1092.491,A -85,B 0,C 180,E1 26432.967,E2 26432.967} C_VEL
LIN {X 0,Y 559.015,Z 1072.618,A -85,B 0,C 180,E1 26431.996,E2 26431.996} C_VEL
LIN {X 0,Y 560.428,Z 1051.647,A -85,B 0,C 180,E1 26431.167,E2 26431.167} C_VEL
LIN {X 0,Y 561.644,Z 1029.692,A -85,B 0,C 180,E1 26430.497,E2 26430.497} C_VEL
LIN {X 0,Y 562.637,Z 1006.33,A -85,B 0,C 180,E1 26429.982,E2 26429.982} C_VEL
LIN {X 0,Y 569.653,Z 754.775,A -85,B 0,C 180,E1 26426.212,E2 26426.212} C_VEL
LIN {X 0,Y 569.964,Z 739.076,A -85,B 0,C 180,E1 26425.96,E2 26425.96} C_VEL
LIN {X 0,Y 564.69,Z 715.782,A -85,B 0,C 180,E1 26425.224,E2 26425.224} C_VEL
LIN {X 0,Y 559.089,Z 704.429,A -85,B 0,C 180,E1 26424.64,E2 26424.64} C_VEL
LIN {X 0,Y 551.626,Z 681.995,A -85,B 0,C 180,E1 26421.954,E2 26421.954} C_VEL
LIN {X 0,Y 545.559,Z 664.713,A -85,B 0,C 180,E1 26419.789,E2 26419.789} C_VEL
LIN {X 0,Y 545.552,Z 664.711,A -85,B 0,C 180,E1 26416.438,E2 26416.438} C_VEL
LIN {X 0,Y 545.562,Z 664.711,A -85,B 0,C 180,E1 26413.129,E2 26413.129} C_VEL
LIN {X 0,Y 545.558,Z 664.71,A -85,B 0,C 180,E1 26409.766,E2 26409.766} C_VEL
LIN {X 0,Y 545.549,Z 664.706,A -85,B 0,C 180,E1 26406.946,E2 26406.946} C_VEL
LIN {X 0,Y 544.559,Z 664.838,A -85,B 0,C 180,E1 26406.137,E2 26406.137} C_VEL
LIN {X 0,Y 538.154,Z 665.63,A -85,B 0,C 180,E1 26403.865,E2 26403.865} C_VEL
LIN {X 0,Y 537.628,Z 665.695,A -85,B 0,C 180,E1 26403.273,E2 26403.273} C_VEL
LIN {X 0,Y 537.616,Z 665.696,A -85,B 0,C 180,E1 26399.898,E2 26399.898} C_VEL
LIN {X 0,Y 537.614,Z 665.698,A -85,B 0,C 180,E1 26396.512,E2 26396.512} C_VEL
LIN {X 0,Y 537.628,Z 665.699,A -85,B 0,C 180,E1 26393.106,E2 26393.106} C_VEL
LIN {X 0,Y 537.619,Z 665.697,A -85,B 0,C 180,E1 26389.56,E2 26389.56} C_VEL
LIN {X 0,Y 537.612,Z 665.702,A -85,B 0,C 180,E1 26386.201,E2 26386.201} C_VEL
LIN {X 0,Y 537.628,Z 665.691,A -85,B 0,C 180,E1 26382.788,E2 26382.788} C_VEL
LIN {X 0,Y 537.619,Z 665.694,A -85,B 0,C 180,E1 26379.313,E2 26379.313} C_VEL
LIN {X 0,Y 537.63,Z 665.701,A -85,B 0,C 180,E1 26375.98,E2 26375.98} C_VEL
LIN {X 0,Y 537.613,Z 665.698,A -85,B 0,C 180,E1 26372.56,E2 26372.56} C_VEL
LIN {X 0,Y 537.619,Z 665.692,A -85,B 0,C 180,E1 26369.149,E2 26369.149} C_VEL
LIN {X 0,Y 537.625,Z 665.69,A -85,B 0,C 180,E1 26365.628,E2 26365.628} C_VEL
LIN {X 0,Y 537.61,Z 665.693,A -85,B 0,C 180,E1 26362.306,E2 26362.306} C_VEL
LIN {X 0,Y 537.61,Z 665.692,A -85,B 0,C 180,E1 26358.957,E2 26358.957} C_VEL
LIN {X 0,Y 537.632,Z 665.693,A -85,B 0,C 180,E1 26355.461,E2 26355.461} C_VEL
LIN {X 0,Y 537.616,Z 665.7,A -85,B 0,C 180,E1 26352.019,E2 26352.019} C_VEL
LIN {X 0,Y 537.613,Z 665.702,A -85,B 0,C 180,E1 26348.623,E2 26348.623} C_VEL
LIN {X 0,Y 537.631,Z 665.696,A -85,B 0,C 180,E1 26345.265,E2 26345.265} C_VEL
LIN {X 0,Y 537.628,Z 665.702,A -85,B 0,C 180,E1 26341.812,E2 26341.812} C_VEL
LIN {X 0,Y 537.622,Z 665.689,A -85,B 0,C 180,E1 26338.369,E2 26338.369} C_VEL
LIN {X 0,Y 537.62,Z 665.694,A -85,B 0,C 180,E1 26334.919,E2 26334.919} C_VEL
LIN {X 0,Y 537.63,Z 665.691,A -85,B 0,C 180,E1 26331.464,E2 26331.464} C_VEL
LIN {X 0,Y 537.634,Z 665.817,A -85,B 0,C 180,E1 26330.159,E2 26330.159} C_VEL
LIN {X 0,Y 546.868,Z 689.88,A -85,B 0,C 180,E1 26327.075,E2 26327.075} C_VEL
LIN {X 0,Y 555.083,Z 712.848,A -85,B 0,C 180,E1 26324.349,E2 26324.349} C_VEL
LIN {X 0,Y 558.056,Z 721.858,A -85,B 0,C 180,E1 26323.33,E2 26323.33} C_VEL
LIN {X 0,Y 555.227,Z 757.921,A -85,B 0,C 180,E1 26320.354,E2 26320.354} C_VEL
LIN {X 0,Y 551.858,Z 802.76,A -85,B 0,C 180,E1 26316.721,E2 26316.721} C_VEL
LIN {X 0,Y 548.723,Z 849.103,A -85,B 0,C 180,E1 26313.014,E2 26313.014} C_VEL
LIN {X 0,Y 545.958,Z 896.589,A -85,B 0,C 180,E1 26309.275,E2 26309.275} C_VEL
LIN {X 0,Y 545.546,Z 905.618,A -85,B 0,C 180,E1 26308.6,E2 26308.6} C_VEL
LIN {X 0,Y 546.454,Z 915.374,A -85,B 0,C 180,E1 26308.382,E2 26308.382} C_VEL
LIN {X 0,Y 542.829,Z 1050.131,A -85,B 0,C 180,E1 26305.928,E2 26305.928} C_VEL
LIN {X 0,Y 542.425,Z 1067.318,A -85,B 0,C 180,E1 26305.417,E2 26305.417} C_VEL
LIN {X 0,Y 541.877,Z 1082.798,A -85,B 0,C 180,E1 26304.763,E2 26304.763} C_VEL
LIN {X 0,Y 541.139,Z 1098.622,A -85,B 0,C 180,E1 26303.87,E2 26303.87} C_VEL
LIN {X 0,Y 540.406,Z 1112.599,A -85,B 0,C 180,E1 26302.865,E2 26302.865} C_VEL
LIN {X 0,Y 539.612,Z 1126.146,A -85,B 0,C 180,E1 26301.638,E2 26301.638} C_VEL
LIN {X 0,Y 538.948,Z 1137.151,A -85,B 0,C 180,E1 26300.413,E2 26300.413} C_VEL
LIN {X 0,Y 538.289,Z 1147.6,A -85,B 0,C 180,E1 26298.97,E2 26298.97} C_VEL
LIN {X 0,Y 537.768,Z 1156.593,A -85,B 0,C 180,E1 26297.419,E2 26297.419} C_VEL
LIN {X 0,Y 537.371,Z 1163.955,A -85,B 0,C 180,E1 26295.763,E2 26295.763} C_VEL
LIN {X 0,Y 537.136,Z 1169.435,A -85,B 0,C 180,E1 26294.115,E2 26294.115} C_VEL
LIN {X 0,Y 537.016,Z 1173.327,A -85,B 0,C 180,E1 26292.364,E2 26292.364} C_VEL
LIN {X 0,Y 537.002,Z 1175.521,A -85,B 0,C 180,E1 26290.553,E2 26290.553} C_VEL
LIN {X 0,Y 537.093,Z 1175.799,A -85,B 0,C 180,E1 26288.781,E2 26288.781} C_VEL
LIN {X 0,Y 537.298,Z 1174.272,A -85,B 0,C 180,E1 26286.948,E2 26286.948} C_VEL
LIN {X 0,Y 537.624,Z 1171.02,A -85,B 0,C 180,E1 26285.229,E2 26285.229} C_VEL
LIN {X 0,Y 538.13,Z 1166.025,A -85,B 0,C 180,E1 26283.515,E2 26283.515} C_VEL
LIN {X 0,Y 538.771,Z 1159.507,A -85,B 0,C 180,E1 26281.914,E2 26281.914} C_VEL
LIN {X 0,Y 539.63,Z 1151.065,A -85,B 0,C 180,E1 26280.319,E2 26280.319} C_VEL
LIN {X 0,Y 540.623,Z 1140.986,A -85,B 0,C 180,E1 26278.834,E2 26278.834} C_VEL
LIN {X 0,Y 541.723,Z 1129.4,A -85,B 0,C 180,E1 26277.461,E2 26277.461} C_VEL
LIN {X 0,Y 542.87,Z 1115.952,A -85,B 0,C 180,E1 26276.198,E2 26276.198} C_VEL
LIN {X 0,Y 543.871,Z 1102.691,A -85,B 0,C 180,E1 26275.202,E2 26275.202} C_VEL
LIN {X 0,Y 544.849,Z 1087.583,A -85,B 0,C 180,E1 26274.313,E2 26274.313} C_VEL
LIN {X 0,Y 545.58,Z 1072.403,A -85,B 0,C 180,E1 26273.634,E2 26273.634} C_VEL
LIN {X 0,Y 546.135,Z 1055.416,A -85,B 0,C 180,E1 26273.089,E2 26273.089} C_VEL
LIN {X 0,Y 549.336,Z 994.949,A -85,B 0,C 180,E1 26271.621,E2 26271.621} C_VEL
LIN {X 0,Y 554.106,Z 919.896,A -85,B 0,C 180,E1 26269.893,E2 26269.893} C_VEL
LIN {X 0,Y 559.49,Z 875.845,A -85,B 0,C 180,E1 26266.02,E2 26266.02} C_VEL
LIN {X 0,Y 565.835,Z 834.429,A -85,B 0,C 180,E1 26262.256,E2 26262.256} C_VEL
LIN {X 0,Y 573.33,Z 795.412,A -85,B 0,C 180,E1 26258.57,E2 26258.57} C_VEL
LIN {X 0,Y 580.249,Z 766.159,A -85,B 0,C 180,E1 26255.679,E2 26255.679} C_VEL
LIN {X 0,Y 582.887,Z 755.55,A -85,B 0,C 180,E1 26254.551,E2 26254.551} C_VEL
LIN {X 0,Y 580.793,Z 746.433,A -85,B 0,C 180,E1 26252.447,E2 26252.447} C_VEL
LIN {X 0,Y 579.322,Z 740.524,A -85,B 0,C 180,E1 26250.642,E2 26250.642} C_VEL
LIN {X 0,Y 578.468,Z 737.03,A -85,B 0,C 180,E1 26249.208,E2 26249.208} C_VEL
LIN {X 0,Y 578.16,Z 735.29,A -85,B 0,C 180,E1 26248.281,E2 26248.281} C_VEL
LIN {X 0,Y 578.285,Z 732.808,A -85,B 0,C 180,E1 26245.913,E2 26245.913} C_VEL
LIN {X 0,Y 578.56,Z 733.22,A -85,B 0,C 180,E1 26244.622,E2 26244.622} C_VEL
LIN {X 0,Y 579.792,Z 736.783,A -85,B 0,C 180,E1 26242.33,E2 26242.33} C_VEL
LIN {X 0,Y 581.154,Z 741.019,A -85,B 0,C 180,E1 26240.844,E2 26240.844} C_VEL
LIN {X 0,Y 582.925,Z 747.153,A -85,B 0,C 180,E1 26239.299,E2 26239.299} C_VEL
LIN {X 0,Y 582.964,Z 748.133,A -85,B 0,C 180,E1 26239.144,E2 26239.144} C_VEL
LIN {X 0,Y 574.398,Z 778.522,A -85,B 0,C 180,E1 26236.686,E2 26236.686} C_VEL
LIN {X 0,Y 568.398,Z 807.965,A -85,B 0,C 180,E1 26234.365,E2 26234.365} C_VEL
LIN {X 0,Y 566.329,Z 829.36,A -85,B 0,C 180,E1 26232.588,E2 26232.588} C_VEL
LIN {X 0,Y 566.601,Z 848.049,A -85,B 0,C 180,E1 26230.948,E2 26230.948} C_VEL
LIN {X 0,Y 569.231,Z 865.82,A -85,B 0,C 180,E1 26229.306,E2 26229.306} C_VEL
LIN {X 0,Y 573.819,Z 881.417,A -85,B 0,C 180,E1 26227.792,E2 26227.792} C_VEL
LIN {X 0,Y 580.263,Z 895.734,A -85,B 0,C 180,E1 26226.351,E2 26226.351} C_VEL
LIN {X 0,Y 588.386,Z 908.649,A -85,B 0,C 180,E1 26225.005,E2 26225.005} C_VEL
LIN {X 0,Y 595.736,Z 918.112,A -85,B 0,C 180,E1 26224.007,E2 26224.007} C_VEL
LIN {X 0,Y 583.766,Z 938.879,A -85,B 0,C 180,E1 26223.352,E2 26223.352} C_VEL
LIN {X 0,Y 574.637,Z 957.867,A -85,B 0,C 180,E1 26222.641,E2 26222.641} C_VEL
LIN {X 0,Y 564.162,Z 981.19,A -85,B 0,C 180,E1 26221.709,E2 26221.709} C_VEL
LIN {X 0,Y 557.749,Z 999.413,A -85,B 0,C 180,E1 26220.908,E2 26220.908} C_VEL
LIN {X 0,Y 555.173,Z 1022.663,A -85,B 0,C 180,E1 26220.662,E2 26220.662} C_VEL
LIN {X 0,Y 553.882,Z 1062.189,A -85,B 0,C 180,E1 26220.042,E2 26220.042} C_VEL
LIN {X 0,Y 552.737,Z 1084.614,A -85,B 0,C 180,E1 26219.507,E2 26219.507} C_VEL
LIN {X 0,Y 551.35,Z 1105.932,A -85,B 0,C 180,E1 26218.81,E2 26218.81} C_VEL
LIN {X 0,Y 549.723,Z 1127.266,A -85,B 0,C 180,E1 26217.926,E2 26217.926} C_VEL
LIN {X 0,Y 548.051,Z 1147.402,A -85,B 0,C 180,E1 26216.9,E2 26216.9} C_VEL
LIN {X 0,Y 546.231,Z 1167.309,A -85,B 0,C 180,E1 26215.668,E2 26215.668} C_VEL
LIN {X 0,Y 544.425,Z 1186.033,A -85,B 0,C 180,E1 26214.291,E2 26214.291} C_VEL
LIN {X 0,Y 542.586,Z 1204.914,A -85,B 0,C 180,E1 26212.651,E2 26212.651} C_VEL
LIN {X 0,Y 541.018,Z 1221.056,A -85,B 0,C 180,E1 26211.009,E2 26211.009} C_VEL
LIN {X 0,Y 539.649,Z 1235.781,A -85,B 0,C 180,E1 26209.255,E2 26209.255} C_VEL
LIN {X 0,Y 538.472,Z 1249.372,A -85,B 0,C 180,E1 26207.359,E2 26207.359} C_VEL
LIN {X 0,Y 537.52,Z 1261.852,A -85,B 0,C 180,E1 26205.315,E2 26205.315} C_VEL
LIN {X 0,Y 536.859,Z 1272.511,A -85,B 0,C 180,E1 26203.242,E2 26203.242} C_VEL
LIN {X 0,Y 536.429,Z 1281.192,A -85,B 0,C 180,E1 26201.176,E2 26201.176} C_VEL
LIN {X 0,Y 536.188,Z 1288.915,A -85,B 0,C 180,E1 26198.902,E2 26198.902} C_VEL
LIN {X 0,Y 536.093,Z 1294.574,A -85,B 0,C 180,E1 26196.746,E2 26196.746} C_VEL
LIN {X 0,Y 536.091,Z 1298.492,A -85,B 0,C 180,E1 26194.599,E2 26194.599} C_VEL
LIN {X 0,Y 536.114,Z 1301.028,A -85,B 0,C 180,E1 26192.35,E2 26192.35} C_VEL
LIN {X 0,Y 536.135,Z 1301.885,A -85,B 0,C 180,E1 26190.212,E2 26190.212} C_VEL
LIN {X 0,Y 536.129,Z 1301.116,A -85,B 0,C 180,E1 26187.968,E2 26187.968} C_VEL
LIN {X 0,Y 536.106,Z 1298.915,A -85,B 0,C 180,E1 26185.827,E2 26185.827} C_VEL
LIN {X 0,Y 536.11,Z 1295.049,A -85,B 0,C 180,E1 26183.681,E2 26183.681} C_VEL
LIN {X 0,Y 536.18,Z 1289.303,A -85,B 0,C 180,E1 26181.419,E2 26181.419} C_VEL
LIN {X 0,Y 536.36,Z 1282.103,A -85,B 0,C 180,E1 26179.249,E2 26179.249} C_VEL
LIN {X 0,Y 536.76,Z 1272.959,A -85,B 0,C 180,E1 26177.082,E2 26177.082} C_VEL
LIN {X 0,Y 537.366,Z 1262.084,A -85,B 0,C 180,E1 26174.955,E2 26174.955} C_VEL
LIN {X 0,Y 538.23,Z 1249.752,A -85,B 0,C 180,E1 26172.93,E2 26172.93} C_VEL
LIN {X 0,Y 539.362,Z 1235.521,A -85,B 0,C 180,E1 26170.956,E2 26170.956} C_VEL
LIN {X 0,Y 540.678,Z 1220.151,A -85,B 0,C 180,E1 26169.151,E2 26169.151} C_VEL
LIN {X 0,Y 542.225,Z 1203.203,A -85,B 0,C 180,E1 26167.444,E2 26167.444} C_VEL
LIN {X 0,Y 543.876,Z 1185.458,A -85,B 0,C 180,E1 26165.911,E2 26165.911} C_VEL
LIN {X 0,Y 545.726,Z 1165.347,A -85,B 0,C 180,E1 26164.437,E2 26164.437} C_VEL
LIN {X 0,Y 547.53,Z 1144.91,A -85,B 0,C 180,E1 26163.187,E2 26163.187} C_VEL
LIN {X 0,Y 549.285,Z 1123.66,A -85,B 0,C 180,E1 26162.105,E2 26162.105} C_VEL
LIN {X 0,Y 551.057,Z 1101.018,A -85,B 0,C 180,E1 26161.17,E2 26161.17} C_VEL
LIN {X 0,Y 552.596,Z 1078.438,A -85,B 0,C 180,E1 26160.434,E2 26160.434} C_VEL
LIN {X 0,Y 554.014,Z 1054.489,A -85,B 0,C 180,E1 26159.858,E2 26159.858} C_VEL
LIN {X 0,Y 555.551,Z 1020.006,A -85,B 0,C 180,E1 26159.274,E2 26159.274} C_VEL
LIN {X 0,Y 557.067,Z 1005.962,A -85,B 0,C 180,E1 26159.082,E2 26159.082} C_VEL
LIN {X 0,Y 566.009,Z 981.527,A -85,B 0,C 180,E1 26157.936,E2 26157.936} C_VEL
LIN {X 0,Y 583.415,Z 944.716,A -85,B 0,C 180,E1 26156.445,E2 26156.445} C_VEL
LIN {X 0,Y 595.111,Z 924.309,A -85,B 0,C 180,E1 26155.756,E2 26155.756} C_VEL
LIN {X 0,Y 597.587,Z 920.13,A -85,B 0,C 180,E1 26155.622,E2 26155.622} C_VEL
LIN {X 0,Y 587.33,Z 906.648,A -85,B 0,C 180,E1 26154.271,E2 26154.271} C_VEL
LIN {X 0,Y 579.076,Z 892.29,A -85,B 0,C 180,E1 26152.915,E2 26152.915} C_VEL
LIN {X 0,Y 572.233,Z 875.553,A -85,B 0,C 180,E1 26151.431,E2 26151.431} C_VEL
LIN {X 0,Y 567.603,Z 858.154,A -85,B 0,C 180,E1 26149.984,E2 26149.984} C_VEL
LIN {X 0,Y 564.889,Z 839.749,A -85,B 0,C 180,E1 26148.546,E2 26148.546} C_VEL
LIN {X 0,Y 564.021,Z 816.991,A -85,B 0,C 180,E1 26146.888,E2 26146.888} C_VEL
LIN {X 0,Y 565.457,Z 790.995,A -85,B 0,C 180,E1 26145.125,E2 26145.125} C_VEL
LIN {X 0,Y 570.123,Z 744.169,A -85,B 0,C 180,E1 26142.034,E2 26142.034} C_VEL
LIN {X 0,Y 570.641,Z 738.648,A -85,B 0,C 180,E1 26141.662,E2 26141.662} C_VEL
LIN {X 0,Y 560.13,Z 714.332,A -85,B 0,C 180,E1 26138.849,E2 26138.849} C_VEL
LIN {X 0,Y 563.426,Z 713.912,A -85,B 0,C 180,E1 26138.17,E2 26138.17} C_VEL
LIN {X 0,Y 564.557,Z 717.753,A -85,B 0,C 180,E1 26137.527,E2 26137.527} C_VEL
LIN {X 0,Y 568.863,Z 727.103,A -85,B 0,C 180,E1 26136.463,E2 26136.463} C_VEL
LIN {X 0,Y 570.588,Z 731.756,A -85,B 0,C 180,E1 26136.055,E2 26136.055} C_VEL
LIN {X 0,Y 572.146,Z 744.363,A -85,B 0,C 180,E1 26135.424,E2 26135.424} C_VEL
LIN {X 0,Y 564.811,Z 835.35,A -85,B 0,C 180,E1 26133.55,E2 26133.55} C_VEL
LIN {X 0,Y 559.639,Z 922.478,A -85,B 0,C 180,E1 26131.872,E2 26131.872} C_VEL
LIN {X 0,Y 555.53,Z 1018.32,A -85,B 0,C 180,E1 26130.151,E2 26130.151} C_VEL
LIN {X 0,Y 554.315,Z 1041.766,A -85,B 0,C 180,E1 26129.524,E2 26129.524} C_VEL
LIN {X 0,Y 552.819,Z 1064.163,A -85,B 0,C 180,E1 26128.726,E2 26128.726} C_VEL
LIN {X 0,Y 551.208,Z 1085.05,A -85,B 0,C 180,E1 26127.788,E2 26127.788} C_VEL
LIN {X 0,Y 549.406,Z 1105.747,A -85,B 0,C 180,E1 26126.655,E2 26126.655} C_VEL
LIN {X 0,Y 547.599,Z 1124.763,A -85,B 0,C 180,E1 26125.411,E2 26125.411} C_VEL
LIN {X 0,Y 545.682,Z 1143.542,A -85,B 0,C 180,E1 26123.946,E2 26123.946} C_VEL
LIN {X 0,Y 543.82,Z 1160.773,A -85,B 0,C 180,E1 26122.355,E2 26122.355} C_VEL
LIN {X 0,Y 542.083,Z 1176.71,A -85,B 0,C 180,E1 26120.629,E2 26120.629} C_VEL
LIN {X 0,Y 540.625,Z 1190.536,A -85,B 0,C 180,E1 26118.885,E2 26118.885} C_VEL
LIN {X 0,Y 539.256,Z 1203.845,A -85,B 0,C 180,E1 26116.907,E2 26116.907} C_VEL
LIN {X 0,Y 538.15,Z 1215.383,A -85,B 0,C 180,E1 26114.857,E2 26114.857} C_VEL
LIN {X 0,Y 537.293,Z 1225.566,A -85,B 0,C 180,E1 26112.685,E2 26112.685} C_VEL
LIN {X 0,Y 536.726,Z 1233.866,A -85,B 0,C 180,E1 26110.519,E2 26110.519} C_VEL
LIN {X 0,Y 536.359,Z 1240.364,A -85,B 0,C 180,E1 26108.361,E2 26108.361} C_VEL
LIN {X 0,Y 536.144,Z 1245.445,A -85,B 0,C 180,E1 26106.102,E2 26106.102} C_VEL
LIN {X 0,Y 536.038,Z 1248.924,A -85,B 0,C 180,E1 26103.85,E2 26103.85} C_VEL
LIN {X 0,Y 536.004,Z 1250.754,A -85,B 0,C 180,E1 26101.603,E2 26101.603} C_VEL
LIN {X 0,Y 536.003,Z 1250.991,A -85,B 0,C 180,E1 26099.359,E2 26099.359} C_VEL
LIN {X 0,Y 536.003,Z 1249.734,A -85,B 0,C 180,E1 26097.113,E2 26097.113} C_VEL
LIN {X 0,Y 536.054,Z 1246.821,A -85,B 0,C 180,E1 26094.863,E2 26094.863} C_VEL
LIN {X 0,Y 536.194,Z 1242.276,A -85,B 0,C 180,E1 26092.607,E2 26092.607} C_VEL
LIN {X 0,Y 536.457,Z 1236.254,A -85,B 0,C 180,E1 26090.401,E2 26090.401} C_VEL
LIN {X 0,Y 536.888,Z 1228.793,A -85,B 0,C 180,E1 26088.288,E2 26088.288} C_VEL
LIN {X 0,Y 537.555,Z 1219.339,A -85,B 0,C 180,E1 26086.116,E2 26086.116} C_VEL
LIN {X 0,Y 538.48,Z 1208.519,A -85,B 0,C 180,E1 26084.049,E2 26084.049} C_VEL
LIN {X 0,Y 539.645,Z 1196.314,A -85,B 0,C 180,E1 26082.087,E2 26082.087} C_VEL
LIN {X 0,Y 541.009,Z 1182.676,A -85,B 0,C 180,E1 26080.231,E2 26080.231} C_VEL
LIN {X 0,Y 542.678,Z 1166.698,A -85,B 0,C 180,E1 26078.377,E2 26078.377} C_VEL
LIN {X 0,Y 544.433,Z 1150.213,A -85,B 0,C 180,E1 26076.742,E2 26076.742} C_VEL
LIN {X 0,Y 546.305,Z 1132.157,A -85,B 0,C 180,E1 26075.22,E2 26075.22} C_VEL
LIN {X 0,Y 548.169,Z 1113.05,A -85,B 0,C 180,E1 26073.863,E2 26073.863} C_VEL
LIN {X 0,Y 549.966,Z 1093.115,A -85,B 0,C 180,E1 26072.673,E2 26072.673} C_VEL
LIN {X 0,Y 551.685,Z 1072.395,A -85,B 0,C 180,E1 26071.65,E2 26071.65} C_VEL
LIN {X 0,Y 553.199,Z 1050.805,A -85,B 0,C 180,E1 26070.79,E2 26070.79} C_VEL
LIN {X 0,Y 554.461,Z 1028.655,A -85,B 0,C 180,E1 26070.117,E2 26070.117} C_VEL
LIN {X 0,Y 555.436,Z 1006.005,A -85,B 0,C 180,E1 26069.619,E2 26069.619} C_VEL
LIN {X 0,Y 562.879,Z 753.006,A -85,B 0,C 180,E1 26065.761,E2 26065.761} C_VEL
LIN {X 0,Y 563.09,Z 740.526,A -85,B 0,C 180,E1 26065.556,E2 26065.556} C_VEL
LIN {X 0,Y 558.381,Z 719.454,A -85,B 0,C 180,E1 26064.876,E2 26064.876} C_VEL
LIN {X 0,Y 551.08,Z 704.867,A -85,B 0,C 180,E1 26064.122,E2 26064.122} C_VEL
LIN {X 0,Y 543.431,Z 682.151,A -85,B 0,C 180,E1 26061.359,E2 26061.359} C_VEL
LIN {X 0,Y 537.613,Z 665.701,A -85,B 0,C 180,E1 26059.281,E2 26059.281} C_VEL
LIN {X 0,Y 537.623,Z 665.702,A -85,B 0,C 180,E1 26055.882,E2 26055.882} C_VEL
LIN {X 0,Y 537.616,Z 665.696,A -85,B 0,C 180,E1 26052.407,E2 26052.407} C_VEL
LIN {X 0,Y 537.612,Z 665.704,A -85,B 0,C 180,E1 26049.088,E2 26049.088} C_VEL
LIN {X 0,Y 537.628,Z 665.701,A -85,B 0,C 180,E1 26045.732,E2 26045.732} C_VEL
LIN {X 0,Y 537.628,Z 665.695,A -85,B 0,C 180,E1 26043.273,E2 26043.273} C_VEL
LIN {X 0,Y 536.64,Z 665.825,A -85,B 0,C 180,E1 26042.452,E2 26042.452} C_VEL
LIN {X 0,Y 530.2,Z 666.621,A -85,B 0,C 180,E1 26040.146,E2 26040.146} C_VEL
LIN {X 0,Y 529.673,Z 666.687,A -85,B 0,C 180,E1 26039.545,E2 26039.545} C_VEL
LIN {X 0,Y 529.682,Z 666.686,A -85,B 0,C 180,E1 26036.095,E2 26036.095} C_VEL
LIN {X 0,Y 529.679,Z 666.688,A -85,B 0,C 180,E1 26032.616,E2 26032.616} C_VEL
LIN {X 0,Y 529.674,Z 666.685,A -85,B 0,C 180,E1 26029.177,E2 26029.177} C_VEL
LIN {X 0,Y 529.684,Z 666.686,A -85,B 0,C 180,E1 26025.69,E2 26025.69} C_VEL
LIN {X 0,Y 529.677,Z 666.683,A -85,B 0,C 180,E1 26022.207,E2 26022.207} C_VEL
LIN {X 0,Y 529.67,Z 666.678,A -85,B 0,C 180,E1 26018.797,E2 26018.797} C_VEL
LIN {X 0,Y 529.679,Z 666.686,A -85,B 0,C 180,E1 26015.417,E2 26015.417} C_VEL
LIN {X 0,Y 529.682,Z 666.69,A -85,B 0,C 180,E1 26011.949,E2 26011.949} C_VEL
LIN {X 0,Y 529.691,Z 666.687,A -85,B 0,C 180,E1 26008.595,E2 26008.595} C_VEL
LIN {X 0,Y 529.687,Z 666.686,A -85,B 0,C 180,E1 26005.02,E2 26005.02} C_VEL
LIN {X 0,Y 529.684,Z 666.685,A -85,B 0,C 180,E1 26001.535,E2 26001.535} C_VEL
LIN {X 0,Y 529.685,Z 666.686,A -85,B 0,C 180,E1 25998.017,E2 25998.017} C_VEL
LIN {X 0,Y 529.684,Z 666.689,A -85,B 0,C 180,E1 25994.565,E2 25994.565} C_VEL
LIN {X 0,Y 529.692,Z 666.692,A -85,B 0,C 180,E1 25991.056,E2 25991.056} C_VEL
LIN {X 0,Y 529.673,Z 666.689,A -85,B 0,C 180,E1 25987.586,E2 25987.586} C_VEL
LIN {X 0,Y 529.681,Z 666.687,A -85,B 0,C 180,E1 25984.149,E2 25984.149} C_VEL
LIN {X 0,Y 529.69,Z 666.686,A -85,B 0,C 180,E1 25980.609,E2 25980.609} C_VEL
LIN {X 0,Y 529.673,Z 666.675,A -85,B 0,C 180,E1 25977.197,E2 25977.197} C_VEL
LIN {X 0,Y 529.678,Z 666.677,A -85,B 0,C 180,E1 25973.784,E2 25973.784} C_VEL
LIN {X 0,Y 529.691,Z 666.726,A -85,B 0,C 180,E1 25970.777,E2 25970.777} C_VEL
LIN {X 0,Y 539.233,Z 691.477,A -85,B 0,C 180,E1 25967.552,E2 25967.552} C_VEL
LIN {X 0,Y 547.38,Z 714.202,A -85,B 0,C 180,E1 25964.795,E2 25964.795} C_VEL
LIN {X 0,Y 550.869,Z 725.288,A -85,B 0,C 180,E1 25963.538,E2 25963.538} C_VEL
LIN {X 0,Y 547.986,Z 760.815,A -85,B 0,C 180,E1 25960.586,E2 25960.586} C_VEL
LIN {X 0,Y 544.454,Z 805.73,A -85,B 0,C 180,E1 25956.908,E2 25956.908} C_VEL
LIN {X 0,Y 541.214,Z 851.797,A -85,B 0,C 180,E1 25953.188,E2 25953.188} C_VEL
LIN {X 0,Y 538.386,Z 898.362,A -85,B 0,C 180,E1 25949.483,E2 25949.483} C_VEL
LIN {X 0,Y 538.013,Z 906.223,A -85,B 0,C 180,E1 25948.891,E2 25948.891} C_VEL
LIN {X 0,Y 538.929,Z 916.202,A -85,B 0,C 180,E1 25948.663,E2 25948.663} C_VEL
LIN {X 0,Y 535.124,Z 1050.673,A -85,B 0,C 180,E1 25946.151,E2 25946.151} C_VEL
LIN {X 0,Y 534.721,Z 1067.338,A -85,B 0,C 180,E1 25945.651,E2 25945.651} C_VEL
LIN {X 0,Y 534.136,Z 1083.377,A -85,B 0,C 180,E1 25944.969,E2 25944.969} C_VEL
LIN {X 0,Y 533.395,Z 1098.751,A -85,B 0,C 180,E1 25944.094,E2 25944.094} C_VEL
LIN {X 0,Y 532.609,Z 1113.249,A -85,B 0,C 180,E1 25943.043,E2 25943.043} C_VEL
LIN {X 0,Y 531.783,Z 1126.823,A -85,B 0,C 180,E1 25941.799,E2 25941.799} C_VEL
LIN {X 0,Y 531.06,Z 1138.315,A -85,B 0,C 180,E1 25940.5,E2 25940.5} C_VEL
LIN {X 0,Y 530.38,Z 1148.716,A -85,B 0,C 180,E1 25939.035,E2 25939.035} C_VEL
LIN {X 0,Y 529.841,Z 1157.67,A -85,B 0,C 180,E1 25937.461,E2 25937.461} C_VEL
LIN {X 0,Y 529.432,Z 1165.007,A -85,B 0,C 180,E1 25935.781,E2 25935.781} C_VEL
LIN {X 0,Y 529.193,Z 1170.466,A -85,B 0,C 180,E1 25934.108,E2 25934.108} C_VEL
LIN {X 0,Y 529.068,Z 1174.385,A -85,B 0,C 180,E1 25932.301,E2 25932.301} C_VEL
LIN {X 0,Y 529.063,Z 1176.548,A -85,B 0,C 180,E1 25930.453,E2 25930.453} C_VEL
LIN {X 0,Y 529.166,Z 1176.791,A -85,B 0,C 180,E1 25928.694,E2 25928.694} C_VEL
LIN {X 0,Y 529.391,Z 1175.267,A -85,B 0,C 180,E1 25926.834,E2 25926.834} C_VEL
LIN {X 0,Y 529.781,Z 1171.75,A -85,B 0,C 180,E1 25924.981,E2 25924.981} C_VEL
LIN {X 0,Y 530.338,Z 1166.634,A -85,B 0,C 180,E1 25923.242,E2 25923.242} C_VEL
LIN {X 0,Y 531.101,Z 1159.446,A -85,B 0,C 180,E1 25921.499,E2 25921.499} C_VEL
LIN {X 0,Y 531.982,Z 1151.439,A -85,B 0,C 180,E1 25920,E2 25920} C_VEL
LIN {X 0,Y 533.119,Z 1140.786,A -85,B 0,C 180,E1 25918.431,E2 25918.431} C_VEL
LIN {X 0,Y 534.244,Z 1129.475,A -85,B 0,C 180,E1 25917.103,E2 25917.103} C_VEL
LIN {X 0,Y 535.423,Z 1116.513,A -85,B 0,C 180,E1 25915.877,E2 25915.877} C_VEL
LIN {X 0,Y 536.479,Z 1103.11,A -85,B 0,C 180,E1 25914.867,E2 25914.867} C_VEL
LIN {X 0,Y 537.532,Z 1088.046,A -85,B 0,C 180,E1 25913.967,E2 25913.967} C_VEL
LIN {X 0,Y 538.338,Z 1072.123,A -85,B 0,C 180,E1 25913.253,E2 25913.253} C_VEL
LIN {X 0,Y 538.901,Z 1056.051,A -85,B 0,C 180,E1 25912.735,E2 25912.735} C_VEL
LIN {X 0,Y 542.176,Z 998.66,A -85,B 0,C 180,E1 25911.287,E2 25911.287} C_VEL
LIN {X 0,Y 547.407,Z 921.324,A -85,B 0,C 180,E1 25909.449,E2 25909.449} C_VEL
LIN {X 0,Y 553.088,Z 877.687,A -85,B 0,C 180,E1 25905.553,E2 25905.553} C_VEL
LIN {X 0,Y 559.551,Z 837.905,A -85,B 0,C 180,E1 25901.885,E2 25901.885} C_VEL
LIN {X 0,Y 567.435,Z 799.225,A -85,B 0,C 180,E1 25898.173,E2 25898.173} C_VEL
LIN {X 0,Y 574.867,Z 769.803,A -85,B 0,C 180,E1 25895.216,E2 25895.216} C_VEL
LIN {X 0,Y 577.399,Z 760.515,A -85,B 0,C 180,E1 25894.218,E2 25894.218} C_VEL
LIN {X 0,Y 575.685,Z 752.288,A -85,B 0,C 180,E1 25892.258,E2 25892.258} C_VEL
LIN {X 0,Y 574.385,Z 746.627,A -85,B 0,C 180,E1 25890.485,E2 25890.485} C_VEL
LIN {X 0,Y 573.69,Z 743.051,A -85,B 0,C 180,E1 25888.942,E2 25888.942} C_VEL
LIN {X 0,Y 573.456,Z 741.646,A -85,B 0,C 180,E1 25888.108,E2 25888.108} C_VEL
LIN {X 0,Y 573.729,Z 739.382,A -85,B 0,C 180,E1 25885.862,E2 25885.862} C_VEL
LIN {X 0,Y 574.008,Z 739.869,A -85,B 0,C 180,E1 25884.606,E2 25884.606} C_VEL
LIN {X 0,Y 575.148,Z 743.327,A -85,B 0,C 180,E1 25882.395,E2 25882.395} C_VEL
LIN {X 0,Y 576.521,Z 747.777,A -85,B 0,C 180,E1 25880.825,E2 25880.825} C_VEL
LIN {X 0,Y 577.806,Z 752.671,A -85,B 0,C 180,E1 25879.586,E2 25879.586} C_VEL
LIN {X 0,Y 569.013,Z 781.665,A -85,B 0,C 180,E1 25877.19,E2 25877.19} C_VEL
LIN {X 0,Y 562.637,Z 810.457,A -85,B 0,C 180,E1 25874.869,E2 25874.869} C_VEL
LIN {X 0,Y 560.207,Z 831.858,A -85,B 0,C 180,E1 25873.053,E2 25873.053} C_VEL
LIN {X 0,Y 560.135,Z 849.999,A -85,B 0,C 180,E1 25871.432,E2 25871.432} C_VEL
LIN {X 0,Y 562.244,Z 867.276,A -85,B 0,C 180,E1 25869.801,E2 25869.801} C_VEL
LIN {X 0,Y 566.159,Z 882.409,A -85,B 0,C 180,E1 25868.306,E2 25868.306} C_VEL
LIN {X 0,Y 572.552,Z 897.899,A -85,B 0,C 180,E1 25866.718,E2 25866.718} C_VEL
LIN {X 0,Y 580.596,Z 911.436,A -85,B 0,C 180,E1 25865.282,E2 25865.282} C_VEL
LIN {X 0,Y 587.056,Z 920.235,A -85,B 0,C 180,E1 25864.344,E2 25864.344} C_VEL
LIN {X 0,Y 575.558,Z 940.784,A -85,B 0,C 180,E1 25863.68,E2 25863.68} C_VEL
LIN {X 0,Y 566.868,Z 959.389,A -85,B 0,C 180,E1 25862.965,E2 25862.965} C_VEL
LIN {X 0,Y 557.733,Z 979.374,A -85,B 0,C 180,E1 25862.169,E2 25862.169} C_VEL
LIN {X 0,Y 550.54,Z 999.406,A -85,B 0,C 180,E1 25861.277,E2 25861.277} C_VEL
LIN {X 0,Y 547.925,Z 1023.308,A -85,B 0,C 180,E1 25861.015,E2 25861.015} C_VEL
LIN {X 0,Y 546.587,Z 1062.453,A -85,B 0,C 180,E1 25860.383,E2 25860.383} C_VEL
LIN {X 0,Y 545.374,Z 1085.212,A -85,B 0,C 180,E1 25859.828,E2 25859.828} C_VEL
LIN {X 0,Y 543.878,Z 1107.083,A -85,B 0,C 180,E1 25859.093,E2 25859.093} C_VEL
LIN {X 0,Y 542.138,Z 1128.817,A -85,B 0,C 180,E1 25858.164,E2 25858.164} C_VEL
LIN {X 0,Y 540.269,Z 1150.035,A -85,B 0,C 180,E1 25857.039,E2 25857.039} C_VEL
LIN {X 0,Y 538.455,Z 1169.317,A -85,B 0,C 180,E1 25855.812,E2 25855.812} C_VEL
LIN {X 0,Y 536.476,Z 1188.879,A -85,B 0,C 180,E1 25854.322,E2 25854.322} C_VEL
LIN {X 0,Y 534.722,Z 1206.089,A -85,B 0,C 180,E1 25852.771,E2 25852.771} C_VEL
LIN {X 0,Y 533.009,Z 1222.955,A -85,B 0,C 180,E1 25850.994,E2 25850.994} C_VEL
LIN {X 0,Y 531.622,Z 1237.462,A -85,B 0,C 180,E1 25849.215,E2 25849.215} C_VEL
LIN {X 0,Y 530.406,Z 1251.295,A -85,B 0,C 180,E1 25847.214,E2 25847.214} C_VEL
LIN {X 0,Y 529.475,Z 1263.054,A -85,B 0,C 180,E1 25845.202,E2 25845.202} C_VEL
LIN {X 0,Y 528.832,Z 1273.371,A -85,B 0,C 180,E1 25843.112,E2 25843.112} C_VEL
LIN {X 0,Y 528.402,Z 1281.909,A -85,B 0,C 180,E1 25841.017,E2 25841.017} C_VEL
LIN {X 0,Y 528.184,Z 1289.066,A -85,B 0,C 180,E1 25838.815,E2 25838.815} C_VEL
LIN {X 0,Y 528.096,Z 1294.57,A -85,B 0,C 180,E1 25836.631,E2 25836.631} C_VEL
LIN {X 0,Y 528.103,Z 1298.401,A -85,B 0,C 180,E1 25834.451,E2 25834.451} C_VEL
LIN {X 0,Y 528.125,Z 1300.769,A -85,B 0,C 180,E1 25832.169,E2 25832.169} C_VEL
LIN {X 0,Y 528.156,Z 1301.533,A -85,B 0,C 180,E1 25829.999,E2 25829.999} C_VEL
LIN {X 0,Y 528.133,Z 1300.652,A -85,B 0,C 180,E1 25827.829,E2 25827.829} C_VEL
LIN {X 0,Y 528.115,Z 1298.173,A -85,B 0,C 180,E1 25825.546,E2 25825.546} C_VEL
LIN {X 0,Y 528.103,Z 1294.186,A -85,B 0,C 180,E1 25823.366,E2 25823.366} C_VEL
LIN {X 0,Y 528.192,Z 1288.541,A -85,B 0,C 180,E1 25821.178,E2 25821.178} C_VEL
LIN {X 0,Y 528.399,Z 1281.232,A -85,B 0,C 180,E1 25818.98,E2 25818.98} C_VEL
LIN {X 0,Y 528.813,Z 1272.306,A -85,B 0,C 180,E1 25816.85,E2 25816.85} C_VEL
LIN {X 0,Y 529.439,Z 1261.858,A -85,B 0,C 180,E1 25814.779,E2 25814.779} C_VEL
LIN {X 0,Y 530.324,Z 1249.927,A -85,B 0,C 180,E1 25812.78,E2 25812.78} C_VEL
LIN {X 0,Y 531.489,Z 1235.958,A -85,B 0,C 180,E1 25810.807,E2 25810.807} C_VEL
LIN {X 0,Y 532.85,Z 1220.938,A -85,B 0,C 180,E1 25808.996,E2 25808.996} C_VEL
LIN {X 0,Y 534.518,Z 1203.735,A -85,B 0,C 180,E1 25807.217,E2 25807.217} C_VEL
LIN {X 0,Y 536.254,Z 1186.188,A -85,B 0,C 180,E1 25805.664,E2 25805.664} C_VEL
LIN {X 0,Y 538.194,Z 1166.176,A -85,B 0,C 180,E1 25804.165,E2 25804.165} C_VEL
LIN {X 0,Y 540.08,Z 1146.154,A -85,B 0,C 180,E1 25802.906,E2 25802.906} C_VEL
LIN {X 0,Y 542.057,Z 1123.913,A -85,B 0,C 180,E1 25801.741,E2 25801.741} C_VEL
LIN {X 0,Y 543.943,Z 1101.393,A -85,B 0,C 180,E1 25800.787,E2 25800.787} C_VEL
LIN {X 0,Y 545.597,Z 1079.076,A -85,B 0,C 180,E1 25800.035,E2 25800.035} C_VEL
LIN {X 0,Y 547.187,Z 1054.324,A -85,B 0,C 180,E1 25799.419,E2 25799.419} C_VEL
LIN {X 0,Y 548.855,Z 1020.268,A -85,B 0,C 180,E1 25798.819,E2 25798.819} C_VEL
LIN {X 0,Y 550.908,Z 1002.107,A -85,B 0,C 180,E1 25798.576,E2 25798.576} C_VEL
LIN {X 0,Y 559.785,Z 978.665,A -85,B 0,C 180,E1 25797.475,E2 25797.475} C_VEL
LIN {X 0,Y 576.953,Z 942.827,A -85,B 0,C 180,E1 25796.019,E2 25796.019} C_VEL
LIN {X 0,Y 588.76,Z 922.073,A -85,B 0,C 180,E1 25795.305,E2 25795.305} C_VEL
LIN {X 0,Y 578.68,Z 907.942,A -85,B 0,C 180,E1 25793.898,E2 25793.898} C_VEL
LIN {X 0,Y 570.811,Z 893.224,A -85,B 0,C 180,E1 25792.516,E2 25792.516} C_VEL
LIN {X 0,Y 564.409,Z 876.441,A -85,B 0,C 180,E1 25791.03,E2 25791.03} C_VEL
LIN {X 0,Y 560.003,Z 858.307,A -85,B 0,C 180,E1 25789.52,E2 25789.52} C_VEL
LIN {X 0,Y 557.585,Z 839.101,A -85,B 0,C 180,E1 25788.018,E2 25788.018} C_VEL
LIN {X 0,Y 557.116,Z 815.418,A -85,B 0,C 180,E1 25786.291,E2 25786.291} C_VEL
LIN {X 0,Y 559.294,Z 785.632,A -85,B 0,C 180,E1 25784.274,E2 25784.274} C_VEL
LIN {X 0,Y 563.84,Z 742.12,A -85,B 0,C 180,E1 25781.366,E2 25781.366} C_VEL
LIN {X 0,Y 555.434,Z 722.551,A -85,B 0,C 180,E1 25779.089,E2 25779.089} C_VEL
LIN {X 0,Y 557.304,Z 722.216,A -85,B 0,C 180,E1 25778.697,E2 25778.697} C_VEL
LIN {X 0,Y 559.748,Z 721.509,A -85,B 0,C 180,E1 25778.229,E2 25778.229} C_VEL
LIN {X 0,Y 563.84,Z 730.474,A -85,B 0,C 180,E1 25777.101,E2 25777.101} C_VEL
LIN {X 0,Y 565.927,Z 736.115,A -85,B 0,C 180,E1 25776.55,E2 25776.55} C_VEL
LIN {X 0,Y 567.021,Z 746.518,A -85,B 0,C 180,E1 25776.018,E2 25776.018} C_VEL
LIN {X 0,Y 559.425,Z 831.632,A -85,B 0,C 180,E1 25774.207,E2 25774.207} C_VEL
LIN {X 0,Y 553.883,Z 913.533,A -85,B 0,C 180,E1 25772.558,E2 25772.558} C_VEL
LIN {X 0,Y 549.83,Z 995.098,A -85,B 0,C 180,E1 25771.052,E2 25771.052} C_VEL
LIN {X 0,Y 548.567,Z 1022.745,A -85,B 0,C 180,E1 25770.497,E2 25770.497} C_VEL
LIN {X 0,Y 547.285,Z 1045.161,A -85,B 0,C 180,E1 25769.859,E2 25769.859} C_VEL
LIN {X 0,Y 545.712,Z 1066.958,A -85,B 0,C 180,E1 25769.049,E2 25769.049} C_VEL
LIN {X 0,Y 543.969,Z 1087.846,A -85,B 0,C 180,E1 25768.071,E2 25768.071} C_VEL
LIN {X 0,Y 542.076,Z 1108.035,A -85,B 0,C 180,E1 25766.926,E2 25766.926} C_VEL
LIN {X 0,Y 540.144,Z 1127.031,A -85,B 0,C 180,E1 25765.641,E2 25765.641} C_VEL
LIN {X 0,Y 538.182,Z 1145.285,A -85,B 0,C 180,E1 25764.183,E2 25764.183} C_VEL
LIN {X 0,Y 536.194,Z 1162.698,A -85,B 0,C 180,E1 25762.533,E2 25762.533} C_VEL
LIN {X 0,Y 534.412,Z 1178.053,A -85,B 0,C 180,E1 25760.824,E2 25760.824} C_VEL
LIN {X 0,Y 532.774,Z 1192.576,A -85,B 0,C 180,E1 25758.933,E2 25758.933} C_VEL
LIN {X 0,Y 531.459,Z 1204.849,A -85,B 0,C 180,E1 25757.068,E2 25757.068} C_VEL
LIN {X 0,Y 530.282,Z 1216.377,A -85,B 0,C 180,E1 25754.971,E2 25754.971} C_VEL
LIN {X 0,Y 529.414,Z 1225.989,A -85,B 0,C 180,E1 25752.877,E2 25752.877} C_VEL
LIN {X 0,Y 528.805,Z 1234.3,A -85,B 0,C 180,E1 25750.679,E2 25750.679} C_VEL
LIN {X 0,Y 528.403,Z 1240.791,A -85,B 0,C 180,E1 25748.488,E2 25748.488} C_VEL
LIN {X 0,Y 528.171,Z 1245.874,A -85,B 0,C 180,E1 25746.195,E2 25746.195} C_VEL
LIN {X 0,Y 528.054,Z 1249.339,A -85,B 0,C 180,E1 25743.909,E2 25743.909} C_VEL
LIN {X 0,Y 528.015,Z 1251.157,A -85,B 0,C 180,E1 25741.628,E2 25741.628} C_VEL
LIN {X 0,Y 528.012,Z 1251.37,A -85,B 0,C 180,E1 25739.349,E2 25739.349} C_VEL
LIN {X 0,Y 528.011,Z 1250.078,A -85,B 0,C 180,E1 25737.069,E2 25737.069} C_VEL
LIN {X 0,Y 528.064,Z 1247.255,A -85,B 0,C 180,E1 25734.867,E2 25734.867} C_VEL
LIN {X 0,Y 528.209,Z 1242.794,A -85,B 0,C 180,E1 25732.604,E2 25732.604} C_VEL
LIN {X 0,Y 528.478,Z 1236.976,A -85,B 0,C 180,E1 25730.416,E2 25730.416} C_VEL
LIN {X 0,Y 528.932,Z 1229.354,A -85,B 0,C 180,E1 25728.219,E2 25728.219} C_VEL
LIN {X 0,Y 529.627,Z 1219.934,A -85,B 0,C 180,E1 25726.016,E2 25726.016} C_VEL
LIN {X 0,Y 530.589,Z 1209.125,A -85,B 0,C 180,E1 25723.917,E2 25723.917} C_VEL
LIN {X 0,Y 531.797,Z 1196.907,A -85,B 0,C 180,E1 25721.927,E2 25721.927} C_VEL
LIN {X 0,Y 533.215,Z 1183.273,A -85,B 0,C 180,E1 25720.045,E2 25720.045} C_VEL
LIN {X 0,Y 534.949,Z 1167.329,A -85,B 0,C 180,E1 25718.164,E2 25718.164} C_VEL
LIN {X 0,Y 536.769,Z 1150.887,A -85,B 0,C 180,E1 25716.507,E2 25716.507} C_VEL
LIN {X 0,Y 538.709,Z 1132.842,A -85,B 0,C 180,E1 25714.964,E2 25714.964} C_VEL
LIN {X 0,Y 540.556,Z 1114.586,A -85,B 0,C 180,E1 25713.644,E2 25713.644} C_VEL
LIN {X 0,Y 542.496,Z 1093.891,A -85,B 0,C 180,E1 25712.384,E2 25712.384} C_VEL
LIN {X 0,Y 544.273,Z 1073.272,A -85,B 0,C 180,E1 25711.348,E2 25711.348} C_VEL
LIN {X 0,Y 545.839,Z 1051.688,A -85,B 0,C 180,E1 25710.474,E2 25710.474} C_VEL
LIN {X 0,Y 547.15,Z 1029.644,A -85,B 0,C 180,E1 25709.789,E2 25709.789} C_VEL
LIN {X 0,Y 548.198,Z 1006.567,A -85,B 0,C 180,E1 25709.27,E2 25709.27} C_VEL
LIN {X 0,Y 555.855,Z 759.484,A -85,B 0,C 180,E1 25705.429,E2 25705.429} C_VEL
LIN {X 0,Y 556.276,Z 742.024,A -85,B 0,C 180,E1 25705.141,E2 25705.141} C_VEL
LIN {X 0,Y 551.978,Z 722.905,A -85,B 0,C 180,E1 25704.515,E2 25704.515} C_VEL
LIN {X 0,Y 542.95,Z 704.936,A -85,B 0,C 180,E1 25703.545,E2 25703.545} C_VEL
LIN {X 0,Y 535.394,Z 682.793,A -85,B 0,C 180,E1 25700.81,E2 25700.81} C_VEL
LIN {X 0,Y 529.689,Z 666.684,A -85,B 0,C 180,E1 25698.755,E2 25698.755} C_VEL
LIN {X 0,Y 529.687,Z 666.688,A -85,B 0,C 180,E1 25695.218,E2 25695.218} C_VEL
LIN {X 0,Y 529.684,Z 666.688,A -85,B 0,C 180,E1 25691.785,E2 25691.785} C_VEL
LIN {X 0,Y 529.683,Z 666.693,A -85,B 0,C 180,E1 25688.252,E2 25688.252} C_VEL
LIN {X 0,Y 529.674,Z 666.69,A -85,B 0,C 180,E1 25684.797,E2 25684.797} C_VEL
LIN {X 0,Y 529.68,Z 666.686,A -85,B 0,C 180,E1 25681.401,E2 25681.401} C_VEL
LIN {X 0,Y 529.673,Z 666.687,A -85,B 0,C 180,E1 25679.545,E2 25679.545} C_VEL
LIN {X 0,Y 528.695,Z 666.812,A -85,B 0,C 180,E1 25678.712,E2 25678.712} C_VEL
LIN {X 0,Y 522.18,Z 667.621,A -85,B 0,C 180,E1 25676.31,E2 25676.31} C_VEL
LIN {X 0,Y 521.743,Z 667.677,A -85,B 0,C 180,E1 25675.761,E2 25675.761} C_VEL
LIN {X 0,Y 521.737,Z 667.679,A -85,B 0,C 180,E1 25672.301,E2 25672.301} C_VEL
LIN {X 0,Y 521.744,Z 667.673,A -85,B 0,C 180,E1 25668.899,E2 25668.899} C_VEL
LIN {X 0,Y 521.738,Z 667.677,A -85,B 0,C 180,E1 25665.337,E2 25665.337} C_VEL
LIN {X 0,Y 521.734,Z 667.672,A -85,B 0,C 180,E1 25661.947,E2 25661.947} C_VEL
LIN {X 0,Y 521.74,Z 667.665,A -85,B 0,C 180,E1 25658.487,E2 25658.487} C_VEL
LIN {X 0,Y 521.737,Z 667.673,A -85,B 0,C 180,E1 25654.949,E2 25654.949} C_VEL
LIN {X 0,Y 521.734,Z 667.677,A -85,B 0,C 180,E1 25651.539,E2 25651.539} C_VEL
LIN {X 0,Y 521.748,Z 667.676,A -85,B 0,C 180,E1 25648.135,E2 25648.135} C_VEL
LIN {X 0,Y 521.74,Z 667.677,A -85,B 0,C 180,E1 25644.613,E2 25644.613} C_VEL
LIN {X 0,Y 521.734,Z 667.68,A -85,B 0,C 180,E1 25641.182,E2 25641.182} C_VEL
LIN {X 0,Y 521.752,Z 667.679,A -85,B 0,C 180,E1 25637.72,E2 25637.72} C_VEL
LIN {X 0,Y 521.743,Z 667.681,A -85,B 0,C 180,E1 25634.211,E2 25634.211} C_VEL
LIN {X 0,Y 521.744,Z 667.678,A -85,B 0,C 180,E1 25630.756,E2 25630.756} C_VEL
LIN {X 0,Y 521.754,Z 667.674,A -85,B 0,C 180,E1 25627.19,E2 25627.19} C_VEL
LIN {X 0,Y 521.75,Z 667.68,A -85,B 0,C 180,E1 25623.726,E2 25623.726} C_VEL
LIN {X 0,Y 521.753,Z 667.676,A -85,B 0,C 180,E1 25620.243,E2 25620.243} C_VEL
LIN {X 0,Y 521.745,Z 667.667,A -85,B 0,C 180,E1 25616.766,E2 25616.766} C_VEL
LIN {X 0,Y 521.745,Z 667.671,A -85,B 0,C 180,E1 25613.233,E2 25613.233} C_VEL
LIN {X 0,Y 521.773,Z 667.805,A -85,B 0,C 180,E1 25611.399,E2 25611.399} C_VEL
LIN {X 0,Y 531.106,Z 691.766,A -85,B 0,C 180,E1 25608.205,E2 25608.205} C_VEL
LIN {X 0,Y 539.036,Z 713.673,A -85,B 0,C 180,E1 25605.482,E2 25605.482} C_VEL
LIN {X 0,Y 543.723,Z 728.084,A -85,B 0,C 180,E1 25603.8,E2 25603.8} C_VEL
LIN {X 0,Y 540.725,Z 763.572,A -85,B 0,C 180,E1 25600.827,E2 25600.827} C_VEL
LIN {X 0,Y 537.142,Z 807.698,A -85,B 0,C 180,E1 25597.185,E2 25597.185} C_VEL
LIN {X 0,Y 533.811,Z 853.126,A -85,B 0,C 180,E1 25593.479,E2 25593.479} C_VEL
LIN {X 0,Y 530.82,Z 900.135,A -85,B 0,C 180,E1 25589.697,E2 25589.697} C_VEL
LIN {X 0,Y 530.507,Z 906.969,A -85,B 0,C 180,E1 25589.187,E2 25589.187} C_VEL
LIN {X 0,Y 531.406,Z 917.169,A -85,B 0,C 180,E1 25588.946,E2 25588.946} C_VEL
LIN {X 0,Y 527.427,Z 1051.35,A -85,B 0,C 180,E1 25586.377,E2 25586.377} C_VEL
LIN {X 0,Y 527.008,Z 1067.885,A -85,B 0,C 180,E1 25585.873,E2 25585.873} C_VEL
LIN {X 0,Y 526.402,Z 1083.941,A -85,B 0,C 180,E1 25585.181,E2 25585.181} C_VEL
LIN {X 0,Y 525.654,Z 1098.931,A -85,B 0,C 180,E1 25584.32,E2 25584.32} C_VEL
LIN {X 0,Y 524.813,Z 1113.854,A -85,B 0,C 180,E1 25583.228,E2 25583.228} C_VEL
LIN {X 0,Y 523.953,Z 1127.471,A -85,B 0,C 180,E1 25581.964,E2 25581.964} C_VEL
LIN {X 0,Y 523.169,Z 1139.43,A -85,B 0,C 180,E1 25580.589,E2 25580.589} C_VEL
LIN {X 0,Y 522.433,Z 1150.333,A -85,B 0,C 180,E1 25579.016,E2 25579.016} C_VEL
LIN {X 0,Y 521.884,Z 1159.06,A -85,B 0,C 180,E1 25577.429,E2 25577.429} C_VEL
LIN {X 0,Y 521.468,Z 1166.446,A -85,B 0,C 180,E1 25575.686,E2 25575.686} C_VEL
LIN {X 0,Y 521.234,Z 1171.759,A -85,B 0,C 180,E1 25573.987,E2 25573.987} C_VEL
LIN {X 0,Y 521.112,Z 1175.703,A -85,B 0,C 180,E1 25572.072,E2 25572.072} C_VEL
LIN {X 0,Y 521.127,Z 1177.594,A -85,B 0,C 180,E1 25570.279,E2 25570.279} C_VEL
LIN {X 0,Y 521.259,Z 1177.714,A -85,B 0,C 180,E1 25568.383,E2 25568.383} C_VEL
LIN {X 0,Y 521.505,Z 1176.09,A -85,B 0,C 180,E1 25566.606,E2 25566.606} C_VEL
LIN {X 0,Y 521.949,Z 1172.49,A -85,B 0,C 180,E1 25564.725,E2 25564.725} C_VEL
LIN {X 0,Y 522.557,Z 1167.243,A -85,B 0,C 180,E1 25562.961,E2 25562.961} C_VEL
LIN {X 0,Y 523.403,Z 1160.055,A -85,B 0,C 180,E1 25561.204,E2 25561.204} C_VEL
LIN {X 0,Y 524.361,Z 1151.839,A -85,B 0,C 180,E1 25559.672,E2 25559.672} C_VEL
LIN {X 0,Y 525.535,Z 1141.571,A -85,B 0,C 180,E1 25558.146,E2 25558.146} C_VEL
LIN {X 0,Y 526.751,Z 1129.997,A -85,B 0,C 180,E1 25556.78,E2 25556.78} C_VEL
LIN {X 0,Y 528.003,Z 1117.13,A -85,B 0,C 180,E1 25555.547,E2 25555.547} C_VEL
LIN {X 0,Y 529.2,Z 1102.929,A -85,B 0,C 180,E1 25554.47,E2 25554.47} C_VEL
LIN {X 0,Y 530.251,Z 1088.616,A -85,B 0,C 180,E1 25553.612,E2 25553.612} C_VEL
LIN {X 0,Y 531.14,Z 1072.008,A -85,B 0,C 180,E1 25552.863,E2 25552.863} C_VEL
LIN {X 0,Y 531.76,Z 1054.686,A -85,B 0,C 180,E1 25552.314,E2 25552.314} C_VEL
LIN {X 0,Y 536.793,Z 978.234,A -85,B 0,C 180,E1 25550.329,E2 25550.329} C_VEL
LIN {X 0,Y 540.803,Z 922.541,A -85,B 0,C 180,E1 25548.968,E2 25548.968} C_VEL
LIN {X 0,Y 546.778,Z 879.398,A -85,B 0,C 180,E1 25545.058,E2 25545.058} C_VEL
LIN {X 0,Y 553.757,Z 839.412,A -85,B 0,C 180,E1 25541.307,E2 25541.307} C_VEL
LIN {X 0,Y 562.123,Z 801.159,A -85,B 0,C 180,E1 25537.57,E2 25537.57} C_VEL
LIN {X 0,Y 569.834,Z 772.656,A -85,B 0,C 180,E1 25534.65,E2 25534.65} C_VEL
LIN {X 0,Y 571.923,Z 765.398,A -85,B 0,C 180,E1 25533.86,E2 25533.86} C_VEL
LIN {X 0,Y 570.531,Z 757.886,A -85,B 0,C 180,E1 25531.986,E2 25531.986} C_VEL
LIN {X 0,Y 569.44,Z 752.362,A -85,B 0,C 180,E1 25530.156,E2 25530.156} C_VEL
LIN {X 0,Y 568.954,Z 748.547,A -85,B 0,C 180,E1 25528.418,E2 25528.418} C_VEL
LIN {X 0,Y 569.141,Z 746.01,A -85,B 0,C 180,E1 25525.914,E2 25525.914} C_VEL
LIN {X 0,Y 569.44,Z 746.357,A -85,B 0,C 180,E1 25524.711,E2 25524.711} C_VEL
LIN {X 0,Y 570.471,Z 749.654,A -85,B 0,C 180,E1 25522.54,E2 25522.54} C_VEL
LIN {X 0,Y 571.738,Z 754.1,A -85,B 0,C 180,E1 25520.937,E2 25520.937} C_VEL
LIN {X 0,Y 572.522,Z 757.866,A -85,B 0,C 180,E1 25519.985,E2 25519.985} C_VEL
LIN {X 0,Y 563.368,Z 786.426,A -85,B 0,C 180,E1 25517.587,E2 25517.587} C_VEL
LIN {X 0,Y 556.859,Z 813.905,A -85,B 0,C 180,E1 25515.318,E2 25515.318} C_VEL
LIN {X 0,Y 554.171,Z 834.767,A -85,B 0,C 180,E1 25513.503,E2 25513.503} C_VEL
LIN {X 0,Y 553.81,Z 853.608,A -85,B 0,C 180,E1 25511.773,E2 25511.773} C_VEL
LIN {X 0,Y 555.951,Z 872.056,A -85,B 0,C 180,E1 25509.988,E2 25509.988} C_VEL
LIN {X 0,Y 560.06,Z 887.787,A -85,B 0,C 180,E1 25508.394,E2 25508.394} C_VEL
LIN {X 0,Y 566.1,Z 902.422,A -85,B 0,C 180,E1 25506.858,E2 25506.858} C_VEL
LIN {X 0,Y 574.038,Z 915.939,A -85,B 0,C 180,E1 25505.394,E2 25505.394} C_VEL
LIN {X 0,Y 578.544,Z 922.359,A -85,B 0,C 180,E1 25504.696,E2 25504.696} C_VEL
LIN {X 0,Y 567.442,Z 942.703,A -85,B 0,C 180,E1 25504.017,E2 25504.017} C_VEL
LIN {X 0,Y 551.038,Z 978.297,A -85,B 0,C 180,E1 25502.608,E2 25502.608} C_VEL
LIN {X 0,Y 543.3,Z 999.67,A -85,B 0,C 180,E1 25501.649,E2 25501.649} C_VEL
LIN {X 0,Y 540.668,Z 1024.157,A -85,B 0,C 180,E1 25501.37,E2 25501.37} C_VEL
LIN {X 0,Y 539.342,Z 1062.074,A -85,B 0,C 180,E1 25500.746,E2 25500.746} C_VEL
LIN {X 0,Y 538.074,Z 1084.896,A -85,B 0,C 180,E1 25500.182,E2 25500.182} C_VEL
LIN {X 0,Y 536.519,Z 1106.812,A -85,B 0,C 180,E1 25499.436,E2 25499.436} C_VEL
LIN {X 0,Y 534.769,Z 1127.82,A -85,B 0,C 180,E1 25498.529,E2 25498.529} C_VEL
LIN {X 0,Y 532.911,Z 1148.315,A -85,B 0,C 180,E1 25497.441,E2 25497.441} C_VEL
LIN {X 0,Y 530.923,Z 1168.545,A -85,B 0,C 180,E1 25496.146,E2 25496.146} C_VEL
LIN {X 0,Y 528.939,Z 1187.473,A -85,B 0,C 180,E1 25494.692,E2 25494.692} C_VEL
LIN {X 0,Y 527.095,Z 1204.896,A -85,B 0,C 180,E1 25493.119,E2 25493.119} C_VEL
LIN {X 0,Y 525.338,Z 1221.564,A -85,B 0,C 180,E1 25491.361,E2 25491.361} C_VEL
LIN {X 0,Y 523.845,Z 1236.585,A -85,B 0,C 180,E1 25489.512,E2 25489.512} C_VEL
LIN {X 0,Y 522.603,Z 1249.754,A -85,B 0,C 180,E1 25487.594,E2 25487.594} C_VEL
LIN {X 0,Y 521.575,Z 1262.266,A -85,B 0,C 180,E1 25485.453,E2 25485.453} C_VEL
LIN {X 0,Y 520.875,Z 1272.752,A -85,B 0,C 180,E1 25483.316,E2 25483.316} C_VEL
LIN {X 0,Y 520.429,Z 1281.341,A -85,B 0,C 180,E1 25481.187,E2 25481.187} C_VEL
LIN {X 0,Y 520.192,Z 1288.555,A -85,B 0,C 180,E1 25478.955,E2 25478.955} C_VEL
LIN {X 0,Y 520.1,Z 1294.121,A -85,B 0,C 180,E1 25476.733,E2 25476.733} C_VEL
LIN {X 0,Y 520.106,Z 1297.974,A -85,B 0,C 180,E1 25474.519,E2 25474.519} C_VEL
LIN {X 0,Y 520.133,Z 1300.37,A -85,B 0,C 180,E1 25472.202,E2 25472.202} C_VEL
LIN {X 0,Y 520.165,Z 1301.14,A -85,B 0,C 180,E1 25469.999,E2 25469.999} C_VEL
LIN {X 0,Y 520.14,Z 1300.268,A -85,B 0,C 180,E1 25467.795,E2 25467.795} C_VEL
LIN {X 0,Y 520.12,Z 1297.959,A -85,B 0,C 180,E1 25465.588,E2 25465.588} C_VEL
LIN {X 0,Y 520.106,Z 1294.007,A -85,B 0,C 180,E1 25463.375,E2 25463.375} C_VEL
LIN {X 0,Y 520.199,Z 1288.124,A -85,B 0,C 180,E1 25461.042,E2 25461.042} C_VEL
LIN {X 0,Y 520.425,Z 1280.785,A -85,B 0,C 180,E1 25458.809,E2 25458.809} C_VEL
LIN {X 0,Y 520.855,Z 1271.99,A -85,B 0,C 180,E1 25456.68,E2 25456.68} C_VEL
LIN {X 0,Y 521.539,Z 1261.357,A -85,B 0,C 180,E1 25454.543,E2 25454.543} C_VEL
LIN {X 0,Y 522.481,Z 1249.397,A -85,B 0,C 180,E1 25452.514,E2 25452.514} C_VEL
LIN {X 0,Y 523.667,Z 1236.016,A -85,B 0,C 180,E1 25450.594,E2 25450.594} C_VEL
LIN {X 0,Y 525.153,Z 1220.64,A -85,B 0,C 180,E1 25448.704,E2 25448.704} C_VEL
LIN {X 0,Y 526.943,Z 1203.155,A -85,B 0,C 180,E1 25446.871,E2 25446.871} C_VEL
LIN {X 0,Y 528.858,Z 1184.911,A -85,B 0,C 180,E1 25445.241,E2 25445.241} C_VEL
LIN {X 0,Y 530.926,Z 1164.935,A -85,B 0,C 180,E1 25443.731,E2 25443.731} C_VEL
LIN {X 0,Y 532.974,Z 1144.411,A -85,B 0,C 180,E1 25442.431,E2 25442.431} C_VEL
LIN {X 0,Y 535.017,Z 1122.828,A -85,B 0,C 180,E1 25441.294,E2 25441.294} C_VEL
LIN {X 0,Y 537.102,Z 1099.196,A -85,B 0,C 180,E1 25440.286,E2 25440.286} C_VEL
LIN {X 0,Y 538.906,Z 1076.273,A -85,B 0,C 180,E1 25439.52,E2 25439.52} C_VEL
LIN {X 0,Y 540.522,Z 1052.717,A -85,B 0,C 180,E1 25438.931,E2 25438.931} C_VEL
LIN {X 0,Y 542.266,Z 1020.222,A -85,B 0,C 180,E1 25438.343,E2 25438.343} C_VEL
LIN {X 0,Y 545.01,Z 997.789,A -85,B 0,C 180,E1 25438.041,E2 25438.041} C_VEL
LIN {X 0,Y 553.246,Z 976.592,A -85,B 0,C 180,E1 25437.042,E2 25437.042} C_VEL
LIN {X 0,Y 570.529,Z 940.907,A -85,B 0,C 180,E1 25435.583,E2 25435.583} C_VEL
LIN {X 0,Y 580.142,Z 924.069,A -85,B 0,C 180,E1 25434.998,E2 25434.998} C_VEL
LIN {X 0,Y 570.113,Z 909.15,A -85,B 0,C 180,E1 25433.518,E2 25433.518} C_VEL
LIN {X 0,Y 562.587,Z 894.036,A -85,B 0,C 180,E1 25432.104,E2 25432.104} C_VEL
LIN {X 0,Y 556.53,Z 876.872,A -85,B 0,C 180,E1 25430.585,E2 25430.585} C_VEL
LIN {X 0,Y 552.389,Z 857.97,A -85,B 0,C 180,E1 25429.01,E2 25429.01} C_VEL
LIN {X 0,Y 550.349,Z 838.368,A -85,B 0,C 180,E1 25427.478,E2 25427.478} C_VEL
LIN {X 0,Y 550.264,Z 814.312,A -85,B 0,C 180,E1 25425.721,E2 25425.721} C_VEL
LIN {X 0,Y 557.021,Z 745.534,A -85,B 0,C 180,E1 25421.058,E2 25421.058} C_VEL
LIN {X 0,Y 551.399,Z 732.142,A -85,B 0,C 180,E1 25419.476,E2 25419.476} C_VEL
LIN {X 0,Y 553.177,Z 731.649,A -85,B 0,C 180,E1 25419.072,E2 25419.072} C_VEL
LIN {X 0,Y 555.043,Z 730.334,A -85,B 0,C 180,E1 25418.735,E2 25418.735} C_VEL
LIN {X 0,Y 557.223,Z 729.721,A -85,B 0,C 180,E1 25418.314,E2 25418.314} C_VEL
LIN {X 0,Y 560.841,Z 738.602,A -85,B 0,C 180,E1 25417.246,E2 25417.246} C_VEL
LIN {X 0,Y 561.54,Z 741.157,A -85,B 0,C 180,E1 25417.027,E2 25417.027} C_VEL
LIN {X 0,Y 562.109,Z 748.708,A -85,B 0,C 180,E1 25416.635,E2 25416.635} C_VEL
LIN {X 0,Y 553.764,Z 834.04,A -85,B 0,C 180,E1 25414.762,E2 25414.762} C_VEL
LIN {X 0,Y 547.457,Z 919.256,A -85,B 0,C 180,E1 25412.991,E2 25412.991} C_VEL
LIN {X 0,Y 543.119,Z 999.202,A -85,B 0,C 180,E1 25411.466,E2 25411.466} C_VEL
LIN {X 0,Y 541.772,Z 1025.663,A -85,B 0,C 180,E1 25410.897,E2 25410.897} C_VEL
LIN {X 0,Y 540.277,Z 1048.765,A -85,B 0,C 180,E1 25410.199,E2 25410.199} C_VEL
LIN {X 0,Y 538.58,Z 1070.484,A -85,B 0,C 180,E1 25409.349,E2 25409.349} C_VEL
LIN {X 0,Y 536.672,Z 1091.889,A -85,B 0,C 180,E1 25408.305,E2 25408.305} C_VEL
LIN {X 0,Y 534.601,Z 1112.262,A -85,B 0,C 180,E1 25407.09,E2 25407.09} C_VEL
LIN {X 0,Y 532.584,Z 1130.596,A -85,B 0,C 180,E1 25405.787,E2 25405.787} C_VEL
LIN {X 0,Y 530.386,Z 1149.442,A -85,B 0,C 180,E1 25404.207,E2 25404.207} C_VEL
LIN {X 0,Y 528.41,Z 1166.065,A -85,B 0,C 180,E1 25402.567,E2 25402.567} C_VEL
LIN {X 0,Y 526.445,Z 1182.236,A -85,B 0,C 180,E1 25400.688,E2 25400.688} C_VEL
LIN {X 0,Y 524.734,Z 1196.426,A -85,B 0,C 180,E1 25398.728,E2 25398.728} C_VEL
LIN {X 0,Y 523.359,Z 1208.491,A -85,B 0,C 180,E1 25396.768,E2 25396.768} C_VEL
LIN {X 0,Y 522.21,Z 1219.571,A -85,B 0,C 180,E1 25394.64,E2 25394.64} C_VEL
LIN {X 0,Y 521.328,Z 1229.182,A -85,B 0,C 180,E1 25392.405,E2 25392.405} C_VEL
LIN {X 0,Y 520.72,Z 1236.844,A -85,B 0,C 180,E1 25390.175,E2 25390.175} C_VEL
LIN {X 0,Y 520.344,Z 1243.119,A -85,B 0,C 180,E1 25387.842,E2 25387.842} C_VEL
LIN {X 0,Y 520.149,Z 1247.695,A -85,B 0,C 180,E1 25385.516,E2 25385.516} C_VEL
LIN {X 0,Y 520.043,Z 1250.523,A -85,B 0,C 180,E1 25383.196,E2 25383.196} C_VEL
LIN {X 0,Y 520.019,Z 1251.787,A -85,B 0,C 180,E1 25380.881,E2 25380.881} C_VEL
LIN {X 0,Y 520.007,Z 1251.584,A -85,B 0,C 180,E1 25378.678,E2 25378.678} C_VEL
LIN {X 0,Y 520.028,Z 1249.7,A -85,B 0,C 180,E1 25376.362,E2 25376.362} C_VEL
LIN {X 0,Y 520.119,Z 1246.058,A -85,B 0,C 180,E1 25373.931,E2 25373.931} C_VEL
LIN {X 0,Y 520.315,Z 1241.217,A -85,B 0,C 180,E1 25371.713,E2 25371.713} C_VEL
LIN {X 0,Y 520.658,Z 1234.63,A -85,B 0,C 180,E1 25369.488,E2 25369.488} C_VEL
LIN {X 0,Y 521.228,Z 1226.359,A -85,B 0,C 180,E1 25367.255,E2 25367.255} C_VEL
LIN {X 0,Y 522.045,Z 1216.796,A -85,B 0,C 180,E1 25365.128,E2 25365.128} C_VEL
LIN {X 0,Y 523.147,Z 1205.171,A -85,B 0,C 180,E1 25362.996,E2 25362.996} C_VEL
LIN {X 0,Y 524.516,Z 1192.117,A -85,B 0,C 180,E1 25360.975,E2 25360.975} C_VEL
LIN {X 0,Y 526.125,Z 1177.633,A -85,B 0,C 180,E1 25359.066,E2 25359.066} C_VEL
LIN {X 0,Y 527.95,Z 1161.7,A -85,B 0,C 180,E1 25357.271,E2 25357.271} C_VEL
LIN {X 0,Y 529.937,Z 1144.075,A -85,B 0,C 180,E1 25355.593,E2 25355.593} C_VEL
LIN {X 0,Y 531.876,Z 1126.147,A -85,B 0,C 180,E1 25354.142,E2 25354.142} C_VEL
LIN {X 0,Y 533.969,Z 1105.828,A -85,B 0,C 180,E1 25352.752,E2 25352.752} C_VEL
LIN {X 0,Y 535.804,Z 1086.522,A -85,B 0,C 180,E1 25351.645,E2 25351.645} C_VEL
LIN {X 0,Y 537.561,Z 1065.297,A -85,B 0,C 180,E1 25350.651,E2 25350.651} C_VEL
LIN {X 0,Y 539.079,Z 1043.759,A -85,B 0,C 180,E1 25349.851,E2 25349.851} C_VEL
LIN {X 0,Y 540.379,Z 1020.289,A -85,B 0,C 180,E1 25349.189,E2 25349.189} C_VEL
LIN {X 0,Y 541.355,Z 996.468,A -85,B 0,C 180,E1 25348.726,E2 25348.726} C_VEL
LIN {X 0,Y 547.923,Z 789.901,A -85,B 0,C 180,E1 25345.479,E2 25345.479} C_VEL
LIN {X 0,Y 549.412,Z 743.461,A -85,B 0,C 180,E1 25344.723,E2 25344.723} C_VEL
LIN {X 0,Y 545.577,Z 726.329,A -85,B 0,C 180,E1 25344.148,E2 25344.148} C_VEL
LIN {X 0,Y 534.836,Z 705.122,A -85,B 0,C 180,E1 25342.968,E2 25342.968} C_VEL
LIN {X 0,Y 527.235,Z 682.892,A -85,B 0,C 180,E1 25340.182,E2 25340.182} C_VEL
LIN {X 0,Y 521.752,Z 667.676,A -85,B 0,C 180,E1 25338.171,E2 25338.171} C_VEL
LIN {X 0,Y 521.746,Z 667.675,A -85,B 0,C 180,E1 25334.684,E2 25334.684} C_VEL
LIN {X 0,Y 521.737,Z 667.684,A -85,B 0,C 180,E1 25331.245,E2 25331.245} C_VEL
LIN {X 0,Y 521.75,Z 667.675,A -85,B 0,C 180,E1 25327.826,E2 25327.826} C_VEL
LIN {X 0,Y 521.743,Z 667.673,A -85,B 0,C 180,E1 25324.311,E2 25324.311} C_VEL
LIN {X 0,Y 521.752,Z 667.67,A -85,B 0,C 180,E1 25320.845,E2 25320.845} C_VEL
LIN {X 0,Y 521.74,Z 667.678,A -85,B 0,C 180,E1 25317.385,E2 25317.385} C_VEL
LIN {X 0,Y 521.743,Z 667.677,A -85,B 0,C 180,E1 25315.761,E2 25315.761} C_VEL
LIN {X 0,Y 520.754,Z 667.805,A -85,B 0,C 180,E1 25314.915,E2 25314.915} C_VEL
LIN {X 0,Y 514.335,Z 668.604,A -85,B 0,C 180,E1 25312.538,E2 25312.538} C_VEL
LIN {X 0,Y 513.81,Z 668.667,A -85,B 0,C 180,E1 25311.918,E2 25311.918} C_VEL
LIN {X 0,Y 513.812,Z 668.667,A -85,B 0,C 180,E1 25308.378,E2 25308.378} C_VEL
LIN {X 0,Y 513.801,Z 668.67,A -85,B 0,C 180,E1 25304.886,E2 25304.886} C_VEL
LIN {X 0,Y 513.808,Z 668.664,A -85,B 0,C 180,E1 25301.337,E2 25301.337} C_VEL
LIN {X 0,Y 513.814,Z 668.656,A -85,B 0,C 180,E1 25297.718,E2 25297.718} C_VEL
LIN {X 0,Y 513.801,Z 668.66,A -85,B 0,C 180,E1 25294.242,E2 25294.242} C_VEL
LIN {X 0,Y 513.801,Z 668.664,A -85,B 0,C 180,E1 25290.671,E2 25290.671} C_VEL
LIN {X 0,Y 513.798,Z 668.669,A -85,B 0,C 180,E1 25287.213,E2 25287.213} C_VEL
LIN {X 0,Y 513.812,Z 668.666,A -85,B 0,C 180,E1 25283.745,E2 25283.745} C_VEL
LIN {X 0,Y 513.798,Z 668.667,A -85,B 0,C 180,E1 25280.254,E2 25280.254} C_VEL
LIN {X 0,Y 513.802,Z 668.667,A -85,B 0,C 180,E1 25276.726,E2 25276.726} C_VEL
LIN {X 0,Y 513.811,Z 668.665,A -85,B 0,C 180,E1 25273.146,E2 25273.146} C_VEL
LIN {X 0,Y 513.796,Z 668.662,A -85,B 0,C 180,E1 25269.721,E2 25269.721} C_VEL
LIN {X 0,Y 513.803,Z 668.667,A -85,B 0,C 180,E1 25266.247,E2 25266.247} C_VEL
LIN {X 0,Y 513.803,Z 668.662,A -85,B 0,C 180,E1 25262.662,E2 25262.662} C_VEL
LIN {X 0,Y 513.798,Z 668.669,A -85,B 0,C 180,E1 25259.217,E2 25259.217} C_VEL
LIN {X 0,Y 513.806,Z 668.672,A -85,B 0,C 180,E1 25255.645,E2 25255.645} C_VEL
LIN {X 0,Y 513.801,Z 668.703,A -85,B 0,C 180,E1 25252.078,E2 25252.078} C_VEL
LIN {X 0,Y 523.119,Z 692.432,A -85,B 0,C 180,E1 25248.819,E2 25248.819} C_VEL
LIN {X 0,Y 531.065,Z 714.153,A -85,B 0,C 180,E1 25246.07,E2 25246.07} C_VEL
LIN {X 0,Y 536.618,Z 730.806,A -85,B 0,C 180,E1 25244.08,E2 25244.08} C_VEL
LIN {X 0,Y 533.467,Z 766.299,A -85,B 0,C 180,E1 25241.075,E2 25241.075} C_VEL
LIN {X 0,Y 529.773,Z 810.085,A -85,B 0,C 180,E1 25237.427,E2 25237.427} C_VEL
LIN {X 0,Y 526.333,Z 855.491,A -85,B 0,C 180,E1 25233.691,E2 25233.691} C_VEL
LIN {X 0,Y 523.263,Z 901.906,A -85,B 0,C 180,E1 25229.917,E2 25229.917} C_VEL
LIN {X 0,Y 522.994,Z 907.617,A -85,B 0,C 180,E1 25229.489,E2 25229.489} C_VEL
LIN {X 0,Y 523.9,Z 918.022,A -85,B 0,C 180,E1 25229.24,E2 25229.24} C_VEL
LIN {X 0,Y 519.738,Z 1050.542,A -85,B 0,C 180,E1 25226.636,E2 25226.636} C_VEL
LIN {X 0,Y 519.343,Z 1066.614,A -85,B 0,C 180,E1 25226.161,E2 25226.161} C_VEL
LIN {X 0,Y 518.708,Z 1083.066,A -85,B 0,C 180,E1 25225.459,E2 25225.459} C_VEL
LIN {X 0,Y 517.96,Z 1098.163,A -85,B 0,C 180,E1 25224.606,E2 25224.606} C_VEL
LIN {X 0,Y 517.094,Z 1112.892,A -85,B 0,C 180,E1 25223.535,E2 25223.535} C_VEL
LIN {X 0,Y 516.24,Z 1126.349,A -85,B 0,C 180,E1 25222.311,E2 25222.311} C_VEL
LIN {X 0,Y 515.396,Z 1138.667,A -85,B 0,C 180,E1 25220.914,E2 25220.914} C_VEL
LIN {X 0,Y 514.651,Z 1149.393,A -85,B 0,C 180,E1 25219.404,E2 25219.404} C_VEL
LIN {X 0,Y 514.047,Z 1158.565,A -85,B 0,C 180,E1 25217.781,E2 25217.781} C_VEL
LIN {X 0,Y 513.624,Z 1165.751,A -85,B 0,C 180,E1 25216.164,E2 25216.164} C_VEL
LIN {X 0,Y 513.316,Z 1171.829,A -85,B 0,C 180,E1 25214.323,E2 25214.323} C_VEL
LIN {X 0,Y 513.184,Z 1175.963,A -85,B 0,C 180,E1 25212.49,E2 25212.49} C_VEL
LIN {X 0,Y 513.171,Z 1178.37,A -85,B 0,C 180,E1 25210.554,E2 25210.554} C_VEL
LIN {X 0,Y 513.292,Z 1178.857,A -85,B 0,C 180,E1 25208.74,E2 25208.74} C_VEL
LIN {X 0,Y 513.548,Z 1177.515,A -85,B 0,C 180,E1 25206.813,E2 25206.813} C_VEL
LIN {X 0,Y 513.956,Z 1174.538,A -85,B 0,C 180,E1 25205.023,E2 25205.023} C_VEL
LIN {X 0,Y 514.616,Z 1169.427,A -85,B 0,C 180,E1 25203.119,E2 25203.119} C_VEL
LIN {X 0,Y 515.406,Z 1163.09,A -85,B 0,C 180,E1 25201.445,E2 25201.445} C_VEL
LIN {X 0,Y 516.445,Z 1154.847,A -85,B 0,C 180,E1 25199.778,E2 25199.778} C_VEL
LIN {X 0,Y 517.641,Z 1145.059,A -85,B 0,C 180,E1 25198.229,E2 25198.229} C_VEL
LIN {X 0,Y 518.95,Z 1133.834,A -85,B 0,C 180,E1 25196.797,E2 25196.797} C_VEL
LIN {X 0,Y 520.25,Z 1121.459,A -85,B 0,C 180,E1 25195.536,E2 25195.536} C_VEL
LIN {X 0,Y 521.497,Z 1108.257,A -85,B 0,C 180,E1 25194.444,E2 25194.444} C_VEL
LIN {X 0,Y 522.644,Z 1094.053,A -85,B 0,C 180,E1 25193.519,E2 25193.519} C_VEL
LIN {X 0,Y 523.619,Z 1079.245,A -85,B 0,C 180,E1 25192.76,E2 25192.76} C_VEL
LIN {X 0,Y 524.349,Z 1063.117,A -85,B 0,C 180,E1 25192.153,E2 25192.153} C_VEL
LIN {X 0,Y 526.61,Z 1024.024,A -85,B 0,C 180,E1 25191.063,E2 25191.063} C_VEL
LIN {X 0,Y 532.963,Z 941.68,A -85,B 0,C 180,E1 25188.937,E2 25188.937} C_VEL
LIN {X 0,Y 534.202,Z 924.061,A -85,B 0,C 180,E1 25188.502,E2 25188.502} C_VEL
LIN {X 0,Y 540.559,Z 881.247,A -85,B 0,C 180,E1 25184.552,E2 25184.552} C_VEL
LIN {X 0,Y 547.815,Z 842.038,A -85,B 0,C 180,E1 25180.82,E2 25180.82} C_VEL
LIN {X 0,Y 556.646,Z 804.179,A -85,B 0,C 180,E1 25177.058,E2 25177.058} C_VEL
LIN {X 0,Y 564.629,Z 776.495,A -85,B 0,C 180,E1 25174.174,E2 25174.174} C_VEL
LIN {X 0,Y 566.56,Z 770.307,A -85,B 0,C 180,E1 25173.475,E2 25173.475} C_VEL
LIN {X 0,Y 565.314,Z 762.914,A -85,B 0,C 180,E1 25171.525,E2 25171.525} C_VEL
LIN {X 0,Y 564.499,Z 757.708,A -85,B 0,C 180,E1 25169.681,E2 25169.681} C_VEL
LIN {X 0,Y 564.159,Z 754.622,A -85,B 0,C 180,E1 25167.999,E2 25167.999} C_VEL
LIN {X 0,Y 564.633,Z 752.542,A -85,B 0,C 180,E1 25165.727,E2 25165.727} C_VEL
LIN {X 0,Y 564.89,Z 753.088,A -85,B 0,C 180,E1 25164.633,E2 25164.633} C_VEL
LIN {X 0,Y 565.872,Z 756.467,A -85,B 0,C 180,E1 25162.499,E2 25162.499} C_VEL
LIN {X 0,Y 567.025,Z 760.65,A -85,B 0,C 180,E1 25160.984,E2 25160.984} C_VEL
LIN {X 0,Y 567.496,Z 762.678,A -85,B 0,C 180,E1 25160.434,E2 25160.434} C_VEL
LIN {X 0,Y 558.137,Z 789.995,A -85,B 0,C 180,E1 25158.093,E2 25158.093} C_VEL
LIN {X 0,Y 551.375,Z 816.433,A -85,B 0,C 180,E1 25155.864,E2 25155.864} C_VEL
LIN {X 0,Y 548.193,Z 837.948,A -85,B 0,C 180,E1 25153.946,E2 25153.946} C_VEL
LIN {X 0,Y 547.566,Z 856.391,A -85,B 0,C 180,E1 25152.218,E2 25152.218} C_VEL
LIN {X 0,Y 549.247,Z 874.227,A -85,B 0,C 180,E1 25150.451,E2 25150.451} C_VEL
LIN {X 0,Y 552.981,Z 890.148,A -85,B 0,C 180,E1 25148.801,E2 25148.801} C_VEL
LIN {X 0,Y 559.173,Z 905.966,A -85,B 0,C 180,E1 25147.106,E2 25147.106} C_VEL
LIN {X 0,Y 567.049,Z 919.786,A -85,B 0,C 180,E1 25145.582,E2 25145.582} C_VEL
LIN {X 0,Y 570.125,Z 924.598,A -85,B 0,C 180,E1 25145.059,E2 25145.059} C_VEL
LIN {X 0,Y 559.552,Z 944.499,A -85,B 0,C 180,E1 25144.377,E2 25144.377} C_VEL
LIN {X 0,Y 543.988,Z 978.393,A -85,B 0,C 180,E1 25143.022,E2 25143.022} C_VEL
LIN {X 0,Y 536.018,Z 1000.262,A -85,B 0,C 180,E1 25142.023,E2 25142.023} C_VEL
LIN {X 0,Y 533.37,Z 1025.781,A -85,B 0,C 180,E1 25141.719,E2 25141.719} C_VEL
LIN {X 0,Y 532.05,Z 1062.369,A -85,B 0,C 180,E1 25141.097,E2 25141.097} C_VEL
LIN {X 0,Y 530.724,Z 1085.197,A -85,B 0,C 180,E1 25140.519,E2 25140.519} C_VEL
LIN {X 0,Y 529.107,Z 1107.114,A -85,B 0,C 180,E1 25139.758,E2 25139.758} C_VEL
LIN {X 0,Y 527.262,Z 1128.377,A -85,B 0,C 180,E1 25138.821,E2 25138.821} C_VEL
LIN {X 0,Y 525.265,Z 1149.45,A -85,B 0,C 180,E1 25137.674,E2 25137.674} C_VEL
LIN {X 0,Y 523.242,Z 1169.263,A -85,B 0,C 180,E1 25136.376,E2 25136.376} C_VEL
LIN {X 0,Y 521.2,Z 1188.119,A -85,B 0,C 180,E1 25134.902,E2 25134.902} C_VEL
LIN {X 0,Y 519.283,Z 1205.513,A -85,B 0,C 180,E1 25133.295,E2 25133.295} C_VEL
LIN {X 0,Y 517.439,Z 1222.316,A -85,B 0,C 180,E1 25131.479,E2 25131.479} C_VEL
LIN {X 0,Y 515.894,Z 1237.263,A -85,B 0,C 180,E1 25129.589,E2 25129.589} C_VEL
LIN {X 0,Y 514.629,Z 1250.365,A -85,B 0,C 180,E1 25127.642,E2 25127.642} C_VEL
LIN {X 0,Y 513.626,Z 1262.135,A -85,B 0,C 180,E1 25125.582,E2 25125.582} C_VEL
LIN {X 0,Y 512.891,Z 1272.693,A -85,B 0,C 180,E1 25123.39,E2 25123.39} C_VEL
LIN {X 0,Y 512.438,Z 1281.182,A -85,B 0,C 180,E1 25121.25,E2 25121.25} C_VEL
LIN {X 0,Y 512.193,Z 1288.427,A -85,B 0,C 180,E1 25118.957,E2 25118.957} C_VEL
LIN {X 0,Y 512.104,Z 1294.088,A -85,B 0,C 180,E1 25116.613,E2 25116.613} C_VEL
LIN {X 0,Y 512.114,Z 1297.701,A -85,B 0,C 180,E1 25114.478,E2 25114.478} C_VEL
LIN {X 0,Y 512.144,Z 1300.033,A -85,B 0,C 180,E1 25112.124,E2 25112.124} C_VEL
LIN {X 0,Y 512.167,Z 1300.755,A -85,B 0,C 180,E1 25109.887,E2 25109.887} C_VEL
LIN {X 0,Y 512.146,Z 1299.804,A -85,B 0,C 180,E1 25107.649,E2 25107.649} C_VEL
LIN {X 0,Y 512.117,Z 1297.227,A -85,B 0,C 180,E1 25105.295,E2 25105.295} C_VEL
LIN {X 0,Y 512.117,Z 1293.154,A -85,B 0,C 180,E1 25103.046,E2 25103.046} C_VEL
LIN {X 0,Y 512.215,Z 1287.387,A -85,B 0,C 180,E1 25100.788,E2 25100.788} C_VEL
LIN {X 0,Y 512.473,Z 1279.922,A -85,B 0,C 180,E1 25098.519,E2 25098.519} C_VEL
LIN {X 0,Y 512.943,Z 1271.048,A -85,B 0,C 180,E1 25096.356,E2 25096.356} C_VEL
LIN {X 0,Y 513.7,Z 1260.262,A -85,B 0,C 180,E1 25094.185,E2 25094.185} C_VEL
LIN {X 0,Y 514.715,Z 1248.164,A -85,B 0,C 180,E1 25092.124,E2 25092.124} C_VEL
LIN {X 0,Y 516.007,Z 1234.695,A -85,B 0,C 180,E1 25090.176,E2 25090.176} C_VEL
LIN {X 0,Y 517.548,Z 1219.707,A -85,B 0,C 180,E1 25088.324,E2 25088.324} C_VEL
LIN {X 0,Y 519.464,Z 1202.073,A -85,B 0,C 180,E1 25086.458,E2 25086.458} C_VEL
LIN {X 0,Y 521.5,Z 1183.75,A -85,B 0,C 180,E1 25084.807,E2 25084.807} C_VEL
LIN {X 0,Y 523.716,Z 1163.749,A -85,B 0,C 180,E1 25083.279,E2 25083.279} C_VEL
LIN {X 0,Y 525.957,Z 1142.604,A -85,B 0,C 180,E1 25081.931,E2 25081.931} C_VEL
LIN {X 0,Y 528.15,Z 1120.861,A -85,B 0,C 180,E1 25080.782,E2 25080.782} C_VEL
LIN {X 0,Y 530.274,Z 1098.057,A -85,B 0,C 180,E1 25079.801,E2 25079.801} C_VEL
LIN {X 0,Y 532.357,Z 1073.594,A -85,B 0,C 180,E1 25078.983,E2 25078.983} C_VEL
LIN {X 0,Y 534.068,Z 1049.398,A -85,B 0,C 180,E1 25078.383,E2 25078.383} C_VEL
LIN {X 0,Y 535.826,Z 1020.113,A -85,B 0,C 180,E1 25077.838,E2 25077.838} C_VEL
LIN {X 0,Y 539.071,Z 994.411,A -85,B 0,C 180,E1 25077.501,E2 25077.501} C_VEL
LIN {X 0,Y 539.662,Z 992.165,A -85,B 0,C 180,E1 25077.435,E2 25077.435} C_VEL
LIN {X 0,Y 547.128,Z 973.607,A -85,B 0,C 180,E1 25076.563,E2 25076.563} C_VEL
LIN {X 0,Y 564.261,Z 938.71,A -85,B 0,C 180,E1 25075.131,E2 25075.131} C_VEL
LIN {X 0,Y 571.495,Z 925.862,A -85,B 0,C 180,E1 25074.672,E2 25074.672} C_VEL
LIN {X 0,Y 561.975,Z 910.902,A -85,B 0,C 180,E1 25073.194,E2 25073.194} C_VEL
LIN {X 0,Y 554.403,Z 894.713,A -85,B 0,C 180,E1 25071.679,E2 25071.679} C_VEL
LIN {X 0,Y 548.824,Z 877.668,A -85,B 0,C 180,E1 25070.168,E2 25070.168} C_VEL
LIN {X 0,Y 544.946,Z 858.305,A -85,B 0,C 180,E1 25068.55,E2 25068.55} C_VEL
LIN {X 0,Y 543.185,Z 837.917,A -85,B 0,C 180,E1 25066.953,E2 25066.953} C_VEL
LIN {X 0,Y 543.434,Z 813.93,A -85,B 0,C 180,E1 25065.194,E2 25065.194} C_VEL
LIN {X 0,Y 550.21,Z 748.941,A -85,B 0,C 180,E1 25060.741,E2 25060.741} C_VEL
LIN {X 0,Y 547.268,Z 741.876,A -85,B 0,C 180,E1 25059.907,E2 25059.907} C_VEL
LIN {X 0,Y 549.185,Z 741.221,A -85,B 0,C 180,E1 25059.451,E2 25059.451} C_VEL
LIN {X 0,Y 550.685,Z 739.899,A -85,B 0,C 180,E1 25059.166,E2 25059.166} C_VEL
LIN {X 0,Y 553.504,Z 738.509,A -85,B 0,C 180,E1 25058.619,E2 25058.619} C_VEL
LIN {X 0,Y 554.621,Z 738.032,A -85,B 0,C 180,E1 25058.412,E2 25058.412} C_VEL
LIN {X 0,Y 557.194,Z 745.273,A -85,B 0,C 180,E1 25057.575,E2 25057.575} C_VEL
LIN {X 0,Y 557.479,Z 750.917,A -85,B 0,C 180,E1 25057.278,E2 25057.278} C_VEL
LIN {X 0,Y 548.386,Z 835.635,A -85,B 0,C 180,E1 25055.362,E2 25055.362} C_VEL
LIN {X 0,Y 541.829,Z 915.236,A -85,B 0,C 180,E1 25053.645,E2 25053.645} C_VEL
LIN {X 0,Y 537.104,Z 991.572,A -85,B 0,C 180,E1 25052.121,E2 25052.121} C_VEL
LIN {X 0,Y 535.431,Z 1022.476,A -85,B 0,C 180,E1 25051.479,E2 25051.479} C_VEL
LIN {X 0,Y 533.929,Z 1045.272,A -85,B 0,C 180,E1 25050.81,E2 25050.81} C_VEL
LIN {X 0,Y 532.057,Z 1067.939,A -85,B 0,C 180,E1 25049.937,E2 25049.937} C_VEL
LIN {X 0,Y 530.081,Z 1088.881,A -85,B 0,C 180,E1 25048.925,E2 25048.925} C_VEL
LIN {X 0,Y 527.99,Z 1108.723,A -85,B 0,C 180,E1 25047.766,E2 25047.766} C_VEL
LIN {X 0,Y 525.726,Z 1128.504,A -85,B 0,C 180,E1 25046.386,E2 25046.386} C_VEL
LIN {X 0,Y 523.481,Z 1147.078,A -85,B 0,C 180,E1 25044.848,E2 25044.848} C_VEL
LIN {X 0,Y 521.275,Z 1164.36,A -85,B 0,C 180,E1 25043.155,E2 25043.155} C_VEL
LIN {X 0,Y 519.239,Z 1180.031,A -85,B 0,C 180,E1 25041.343,E2 25041.343} C_VEL
LIN {X 0,Y 517.425,Z 1194.272,A -85,B 0,C 180,E1 25039.413,E2 25039.413} C_VEL
LIN {X 0,Y 515.94,Z 1206.484,A -85,B 0,C 180,E1 25037.481,E2 25037.481} C_VEL
LIN {X 0,Y 514.625,Z 1217.92,A -85,B 0,C 180,E1 25035.322,E2 25035.322} C_VEL
LIN {X 0,Y 513.645,Z 1227.403,A -85,B 0,C 180,E1 25033.165,E2 25033.165} C_VEL
LIN {X 0,Y 512.948,Z 1235.582,A -85,B 0,C 180,E1 25030.899,E2 25030.899} C_VEL
LIN {X 0,Y 512.478,Z 1242.316,A -85,B 0,C 180,E1 25028.527,E2 25028.527} C_VEL
LIN {X 0,Y 512.213,Z 1247.17,A -85,B 0,C 180,E1 25026.163,E2 25026.163} C_VEL
LIN {X 0,Y 512.076,Z 1250.522,A -85,B 0,C 180,E1 25023.695,E2 25023.695} C_VEL
LIN {X 0,Y 512.031,Z 1252.123,A -85,B 0,C 180,E1 25021.343,E2 25021.343} C_VEL
LIN {X 0,Y 512.023,Z 1252.055,A -85,B 0,C 180,E1 25019.024,E2 25019.024} C_VEL
LIN {X 0,Y 512.029,Z 1250.395,A -85,B 0,C 180,E1 25016.641,E2 25016.641} C_VEL
LIN {X 0,Y 512.119,Z 1247.192,A -85,B 0,C 180,E1 25014.285,E2 25014.285} C_VEL
LIN {X 0,Y 512.285,Z 1242.503,A -85,B 0,C 180,E1 25012.034,E2 25012.034} C_VEL
LIN {X 0,Y 512.638,Z 1235.879,A -85,B 0,C 180,E1 25009.663,E2 25009.663} C_VEL
LIN {X 0,Y 513.216,Z 1227.841,A -85,B 0,C 180,E1 25007.396,E2 25007.396} C_VEL
LIN {X 0,Y 514.05,Z 1218.136,A -85,B 0,C 180,E1 25005.18,E2 25005.18} C_VEL
LIN {X 0,Y 515.134,Z 1207.009,A -85,B 0,C 180,E1 25003.073,E2 25003.073} C_VEL
LIN {X 0,Y 516.604,Z 1193.436,A -85,B 0,C 180,E1 25000.907,E2 25000.907} C_VEL
LIN {X 0,Y 518.255,Z 1179.12,A -85,B 0,C 180,E1 24998.97,E2 24998.97} C_VEL
LIN {X 0,Y 520.127,Z 1163.304,A -85,B 0,C 180,E1 24997.15,E2 24997.15} C_VEL
LIN {X 0,Y 522.092,Z 1146.427,A -85,B 0,C 180,E1 24995.498,E2 24995.498} C_VEL
LIN {X 0,Y 524.227,Z 1127.529,A -85,B 0,C 180,E1 24993.925,E2 24993.925} C_VEL
LIN {X 0,Y 526.3,Z 1108.21,A -85,B 0,C 180,E1 24992.567,E2 24992.567} C_VEL
LIN {X 0,Y 528.277,Z 1088.195,A -85,B 0,C 180,E1 24991.389,E2 24991.389} C_VEL
LIN {X 0,Y 530.075,Z 1067.193,A -85,B 0,C 180,E1 24990.382,E2 24990.382} C_VEL
LIN {X 0,Y 531.698,Z 1045.276,A -85,B 0,C 180,E1 24989.542,E2 24989.542} C_VEL
LIN {X 0,Y 533.016,Z 1023.078,A -85,B 0,C 180,E1 24988.889,E2 24988.889} C_VEL
LIN {X 0,Y 534.039,Z 1000.162,A -85,B 0,C 180,E1 24988.413,E2 24988.413} C_VEL
LIN {X 0,Y 540.847,Z 795.747,A -85,B 0,C 180,E1 24985.139,E2 24985.139} C_VEL
LIN {X 0,Y 542.632,Z 745.03,A -85,B 0,C 180,E1 24984.297,E2 24984.297} C_VEL
LIN {X 0,Y 539.268,Z 730.025,A -85,B 0,C 180,E1 24983.785,E2 24983.785} C_VEL
LIN {X 0,Y 526.836,Z 705.562,A -85,B 0,C 180,E1 24982.41,E2 24982.41} C_VEL
LIN {X 0,Y 519.217,Z 683.578,A -85,B 0,C 180,E1 24979.61,E2 24979.61} C_VEL
LIN {X 0,Y 513.802,Z 668.669,A -85,B 0,C 180,E1 24977.637,E2 24977.637} C_VEL
LIN {X 0,Y 513.796,Z 668.668,A -85,B 0,C 180,E1 24974.164,E2 24974.164} C_VEL
LIN {X 0,Y 513.813,Z 668.667,A -85,B 0,C 180,E1 24970.628,E2 24970.628} C_VEL
LIN {X 0,Y 513.796,Z 668.661,A -85,B 0,C 180,E1 24967.07,E2 24967.07} C_VEL
LIN {X 0,Y 513.801,Z 668.663,A -85,B 0,C 180,E1 24963.6,E2 24963.6} C_VEL
LIN {X 0,Y 513.806,Z 668.662,A -85,B 0,C 180,E1 24960.003,E2 24960.003} C_VEL
LIN {X 0,Y 513.798,Z 668.665,A -85,B 0,C 180,E1 24956.591,E2 24956.591} C_VEL
LIN {X 0,Y 513.812,Z 668.666,A -85,B 0,C 180,E1 24953.149,E2 24953.149} C_VEL
LIN {X 0,Y 513.81,Z 668.667,A -85,B 0,C 180,E1 24951.918,E2 24951.918} C_VEL
LIN {X 0,Y 512.829,Z 668.789,A -85,B 0,C 180,E1 24951.059,E2 24951.059} C_VEL
LIN {X 0,Y 506.304,Z 669.606,A -85,B 0,C 180,E1 24948.583,E2 24948.583} C_VEL
LIN {X 0,Y 505.866,Z 669.656,A -85,B 0,C 180,E1 24948.016,E2 24948.016} C_VEL
LIN {X 0,Y 505.865,Z 669.65,A -85,B 0,C 180,E1 24944.411,E2 24944.411} C_VEL
LIN {X 0,Y 505.87,Z 669.657,A -85,B 0,C 180,E1 24940.94,E2 24940.94} C_VEL
LIN {X 0,Y 505.876,Z 669.652,A -85,B 0,C 180,E1 24937.269,E2 24937.269} C_VEL
LIN {X 0,Y 505.858,Z 669.648,A -85,B 0,C 180,E1 24933.741,E2 24933.741} C_VEL
LIN {X 0,Y 505.879,Z 669.645,A -85,B 0,C 180,E1 24930.228,E2 24930.228} C_VEL
LIN {X 0,Y 505.862,Z 669.65,A -85,B 0,C 180,E1 24926.716,E2 24926.716} C_VEL
LIN {X 0,Y 505.86,Z 669.652,A -85,B 0,C 180,E1 24923.191,E2 24923.191} C_VEL
LIN {X 0,Y 505.866,Z 669.651,A -85,B 0,C 180,E1 24919.64,E2 24919.64} C_VEL
LIN {X 0,Y 505.874,Z 669.651,A -85,B 0,C 180,E1 24916.165,E2 24916.165} C_VEL
LIN {X 0,Y 505.872,Z 669.652,A -85,B 0,C 180,E1 24912.637,E2 24912.637} C_VEL
LIN {X 0,Y 505.868,Z 669.654,A -85,B 0,C 180,E1 24909.16,E2 24909.16} C_VEL
LIN {X 0,Y 505.869,Z 669.657,A -85,B 0,C 180,E1 24905.673,E2 24905.673} C_VEL
LIN {X 0,Y 505.866,Z 669.653,A -85,B 0,C 180,E1 24902.196,E2 24902.196} C_VEL
LIN {X 0,Y 505.877,Z 669.645,A -85,B 0,C 180,E1 24898.636,E2 24898.636} C_VEL
LIN {X 0,Y 505.861,Z 669.65,A -85,B 0,C 180,E1 24895.028,E2 24895.028} C_VEL
LIN {X 0,Y 505.894,Z 669.794,A -85,B 0,C 180,E1 24892.739,E2 24892.739} C_VEL
LIN {X 0,Y 514.507,Z 691.544,A -85,B 0,C 180,E1 24889.676,E2 24889.676} C_VEL
LIN {X 0,Y 522.239,Z 712.324,A -85,B 0,C 180,E1 24886.959,E2 24886.959} C_VEL
LIN {X 0,Y 529.49,Z 733.765,A -85,B 0,C 180,E1 24884.349,E2 24884.349} C_VEL
LIN {X 0,Y 526.273,Z 768.568,A -85,B 0,C 180,E1 24881.371,E2 24881.371} C_VEL
LIN {X 0,Y 522.431,Z 812.157,A -85,B 0,C 180,E1 24877.698,E2 24877.698} C_VEL
LIN {X 0,Y 518.903,Z 856.957,A -85,B 0,C 180,E1 24873.974,E2 24873.974} C_VEL
LIN {X 0,Y 515.705,Z 903.635,A -85,B 0,C 180,E1 24870.144,E2 24870.144} C_VEL
LIN {X 0,Y 515.49,Z 908.289,A -85,B 0,C 180,E1 24869.797,E2 24869.797} C_VEL
LIN {X 0,Y 516.398,Z 918.89,A -85,B 0,C 180,E1 24869.54,E2 24869.54} C_VEL
LIN {X 0,Y 512.028,Z 1051.246,A -85,B 0,C 180,E1 24866.864,E2 24866.864} C_VEL
LIN {X 0,Y 511.618,Z 1067.272,A -85,B 0,C 180,E1 24866.382,E2 24866.382} C_VEL
LIN {X 0,Y 510.975,Z 1083.387,A -85,B 0,C 180,E1 24865.686,E2 24865.686} C_VEL
LIN {X 0,Y 510.182,Z 1098.916,A -85,B 0,C 180,E1 24864.798,E2 24864.798} C_VEL
LIN {X 0,Y 509.259,Z 1114.092,A -85,B 0,C 180,E1 24863.673,E2 24863.673} C_VEL
LIN {X 0,Y 508.373,Z 1127.517,A -85,B 0,C 180,E1 24862.426,E2 24862.426} C_VEL
LIN {X 0,Y 507.477,Z 1140.239,A -85,B 0,C 180,E1 24860.951,E2 24860.951} C_VEL
LIN {X 0,Y 506.708,Z 1150.894,A -85,B 0,C 180,E1 24859.404,E2 24859.404} C_VEL
LIN {X 0,Y 506.083,Z 1160.187,A -85,B 0,C 180,E1 24857.714,E2 24857.714} C_VEL
LIN {X 0,Y 505.627,Z 1167.616,A -85,B 0,C 180,E1 24855.955,E2 24855.955} C_VEL
LIN {X 0,Y 505.35,Z 1173.48,A -85,B 0,C 180,E1 24854.086,E2 24854.086} C_VEL
LIN {X 0,Y 505.22,Z 1177.522,A -85,B 0,C 180,E1 24852.11,E2 24852.11} C_VEL
LIN {X 0,Y 505.245,Z 1179.536,A -85,B 0,C 180,E1 24850.26,E2 24850.26} C_VEL
LIN {X 0,Y 505.399,Z 1179.758,A -85,B 0,C 180,E1 24848.304,E2 24848.304} C_VEL
LIN {X 0,Y 505.695,Z 1178.282,A -85,B 0,C 180,E1 24846.471,E2 24846.471} C_VEL
LIN {X 0,Y 506.203,Z 1174.812,A -85,B 0,C 180,E1 24844.532,E2 24844.532} C_VEL
LIN {X 0,Y 506.901,Z 1169.727,A -85,B 0,C 180,E1 24842.713,E2 24842.713} C_VEL
LIN {X 0,Y 507.853,Z 1162.684,A -85,B 0,C 180,E1 24840.903,E2 24840.903} C_VEL
LIN {X 0,Y 508.96,Z 1154.533,A -85,B 0,C 180,E1 24839.294,E2 24839.294} C_VEL
LIN {X 0,Y 510.354,Z 1143.917,A -85,B 0,C 180,E1 24837.642,E2 24837.642} C_VEL
LIN {X 0,Y 511.774,Z 1132.085,A -85,B 0,C 180,E1 24836.191,E2 24836.191} C_VEL
LIN {X 0,Y 513.125,Z 1119.799,A -85,B 0,C 180,E1 24834.969,E2 24834.969} C_VEL
LIN {X 0,Y 514.544,Z 1105.149,A -85,B 0,C 180,E1 24833.809,E2 24833.809} C_VEL
LIN {X 0,Y 515.722,Z 1091.066,A -85,B 0,C 180,E1 24832.928,E2 24832.928} C_VEL
LIN {X 0,Y 516.784,Z 1074.368,A -85,B 0,C 180,E1 24832.132,E2 24832.132} C_VEL
LIN {X 0,Y 517.612,Z 1055.258,A -85,B 0,C 180,E1 24831.496,E2 24831.496} C_VEL
LIN {X 0,Y 523.593,Z 977.646,A -85,B 0,C 180,E1 24829.337,E2 24829.337} C_VEL
LIN {X 0,Y 527.75,Z 925.51,A -85,B 0,C 180,E1 24827.999,E2 24827.999} C_VEL
LIN {X 0,Y 534.308,Z 883.71,A -85,B 0,C 180,E1 24824.088,E2 24824.088} C_VEL
LIN {X 0,Y 541.992,Z 844.867,A -85,B 0,C 180,E1 24820.325,E2 24820.325} C_VEL
LIN {X 0,Y 550.879,Z 808.858,A -85,B 0,C 180,E1 24816.691,E2 24816.691} C_VEL
LIN {X 0,Y 559.268,Z 781.416,A -85,B 0,C 180,E1 24813.794,E2 24813.794} C_VEL
LIN {X 0,Y 561.222,Z 775.285,A -85,B 0,C 180,E1 24813.093,E2 24813.093} C_VEL
LIN {X 0,Y 560.25,Z 768.035,A -85,B 0,C 180,E1 24811.075,E2 24811.075} C_VEL
LIN {X 0,Y 559.645,Z 763.188,A -85,B 0,C 180,E1 24809.151,E2 24809.151} C_VEL
LIN {X 0,Y 559.47,Z 760.974,A -85,B 0,C 180,E1 24807.819,E2 24807.819} C_VEL
LIN {X 0,Y 560.146,Z 759.162,A -85,B 0,C 180,E1 24805.538,E2 24805.538} C_VEL
LIN {X 0,Y 560.343,Z 759.82,A -85,B 0,C 180,E1 24804.554,E2 24804.554} C_VEL
LIN {X 0,Y 561.221,Z 762.941,A -85,B 0,C 180,E1 24802.588,E2 24802.588} C_VEL
LIN {X 0,Y 562.24,Z 766.961,A -85,B 0,C 180,E1 24801.113,E2 24801.113} C_VEL
LIN {X 0,Y 562.294,Z 768.194,A -85,B 0,C 180,E1 24800.83,E2 24800.83} C_VEL
LIN {X 0,Y 552.236,Z 796.21,A -85,B 0,C 180,E1 24798.396,E2 24798.396} C_VEL
LIN {X 0,Y 545.253,Z 822.598,A -85,B 0,C 180,E1 24796.108,E2 24796.108} C_VEL
LIN {X 0,Y 542.112,Z 843.396,A -85,B 0,C 180,E1 24794.199,E2 24794.199} C_VEL
LIN {X 0,Y 541.439,Z 862.18,A -85,B 0,C 180,E1 24792.378,E2 24792.378} C_VEL
LIN {X 0,Y 543.268,Z 880.433,A -85,B 0,C 180,E1 24790.516,E2 24790.516} C_VEL
LIN {X 0,Y 547.05,Z 895.933,A -85,B 0,C 180,E1 24788.864,E2 24788.864} C_VEL
LIN {X 0,Y 553.225,Z 911.484,A -85,B 0,C 180,E1 24787.15,E2 24787.15} C_VEL
LIN {X 0,Y 561.503,Z 925.787,A -85,B 0,C 180,E1 24785.531,E2 24785.531} C_VEL
LIN {X 0,Y 561.998,Z 926.515,A -85,B 0,C 180,E1 24785.449,E2 24785.449} C_VEL
LIN {X 0,Y 551.307,Z 947.225,A -85,B 0,C 180,E1 24784.712,E2 24784.712} C_VEL
LIN {X 0,Y 537.326,Z 977.645,A -85,B 0,C 180,E1 24783.484,E2 24783.484} C_VEL
LIN {X 0,Y 528.677,Z 1001.318,A -85,B 0,C 180,E1 24782.398,E2 24782.398} C_VEL
LIN {X 0,Y 526.118,Z 1026.803,A -85,B 0,C 180,E1 24782.082,E2 24782.082} C_VEL
LIN {X 0,Y 524.802,Z 1062.159,A -85,B 0,C 180,E1 24781.467,E2 24781.467} C_VEL
LIN {X 0,Y 523.422,Z 1085.002,A -85,B 0,C 180,E1 24780.88,E2 24780.88} C_VEL
LIN {X 0,Y 521.765,Z 1106.686,A -85,B 0,C 180,E1 24780.116,E2 24780.116} C_VEL
LIN {X 0,Y 519.838,Z 1128.089,A -85,B 0,C 180,E1 24779.161,E2 24779.161} C_VEL
LIN {X 0,Y 517.747,Z 1149.363,A -85,B 0,C 180,E1 24777.986,E2 24777.986} C_VEL
LIN {X 0,Y 515.648,Z 1169.127,A -85,B 0,C 180,E1 24776.671,E2 24776.671} C_VEL
LIN {X 0,Y 513.536,Z 1187.967,A -85,B 0,C 180,E1 24775.176,E2 24775.176} C_VEL
LIN {X 0,Y 511.547,Z 1205.349,A -85,B 0,C 180,E1 24773.547,E2 24773.547} C_VEL
LIN {X 0,Y 509.636,Z 1222.164,A -85,B 0,C 180,E1 24771.703,E2 24771.703} C_VEL
LIN {X 0,Y 508.035,Z 1237.114,A -85,B 0,C 180,E1 24769.785,E2 24769.785} C_VEL
LIN {X 0,Y 506.655,Z 1250.961,A -85,B 0,C 180,E1 24767.691,E2 24767.691} C_VEL
LIN {X 0,Y 505.629,Z 1262.573,A -85,B 0,C 180,E1 24765.599,E2 24765.599} C_VEL
LIN {X 0,Y 504.864,Z 1273.373,A -85,B 0,C 180,E1 24763.28,E2 24763.28} C_VEL
LIN {X 0,Y 504.41,Z 1281.814,A -85,B 0,C 180,E1 24761.084,E2 24761.084} C_VEL
LIN {X 0,Y 504.186,Z 1288.765,A -85,B 0,C 180,E1 24758.782,E2 24758.782} C_VEL
LIN {X 0,Y 504.111,Z 1294.256,A -85,B 0,C 180,E1 24756.376,E2 24756.376} C_VEL
LIN {X 0,Y 504.125,Z 1297.889,A -85,B 0,C 180,E1 24754.093,E2 24754.093} C_VEL
LIN {X 0,Y 504.162,Z 1299.823,A -85,B 0,C 180,E1 24751.817,E2 24751.817} C_VEL
LIN {X 0,Y 504.17,Z 1300.258,A -85,B 0,C 180,E1 24749.43,E2 24749.43} C_VEL
LIN {X 0,Y 504.156,Z 1299.18,A -85,B 0,C 180,E1 24747.27,E2 24747.27} C_VEL
LIN {X 0,Y 504.118,Z 1296.319,A -85,B 0,C 180,E1 24744.878,E2 24744.878} C_VEL
LIN {X 0,Y 504.146,Z 1292.035,A -85,B 0,C 180,E1 24742.592,E2 24742.592} C_VEL
LIN {X 0,Y 504.255,Z 1285.999,A -85,B 0,C 180,E1 24740.295,E2 24740.295} C_VEL
LIN {X 0,Y 504.576,Z 1278.205,A -85,B 0,C 180,E1 24737.989,E2 24737.989} C_VEL
LIN {X 0,Y 505.117,Z 1269.103,A -85,B 0,C 180,E1 24735.79,E2 24735.79} C_VEL
LIN {X 0,Y 505.98,Z 1257.985,A -85,B 0,C 180,E1 24733.584,E2 24733.584} C_VEL
LIN {X 0,Y 507.127,Z 1245.469,A -85,B 0,C 180,E1 24731.491,E2 24731.491} C_VEL
LIN {X 0,Y 508.558,Z 1231.658,A -85,B 0,C 180,E1 24729.513,E2 24729.513} C_VEL
LIN {X 0,Y 510.306,Z 1215.966,A -85,B 0,C 180,E1 24727.597,E2 24727.597} C_VEL
LIN {X 0,Y 512.24,Z 1199.304,A -85,B 0,C 180,E1 24725.86,E2 24725.86} C_VEL
LIN {X 0,Y 514.437,Z 1180.596,A -85,B 0,C 180,E1 24724.189,E2 24724.189} C_VEL
LIN {X 0,Y 516.73,Z 1161.009,A -85,B 0,C 180,E1 24722.702,E2 24722.702} C_VEL
LIN {X 0,Y 519.048,Z 1140.65,A -85,B 0,C 180,E1 24721.398,E2 24721.398} C_VEL
LIN {X 0,Y 521.316,Z 1119.51,A -85,B 0,C 180,E1 24720.276,E2 24720.276} C_VEL
LIN {X 0,Y 523.593,Z 1096.55,A -85,B 0,C 180,E1 24719.279,E2 24719.279} C_VEL
LIN {X 0,Y 525.79,Z 1072.577,A -85,B 0,C 180,E1 24718.468,E2 24718.468} C_VEL
LIN {X 0,Y 527.7,Z 1047.14,A -85,B 0,C 180,E1 24717.828,E2 24717.828} C_VEL
LIN {X 0,Y 529.504,Z 1019.955,A -85,B 0,C 180,E1 24717.311,E2 24717.311} C_VEL
LIN {X 0,Y 532.882,Z 994.037,A -85,B 0,C 180,E1 24716.96,E2 24716.96} C_VEL
LIN {X 0,Y 534.007,Z 987.339,A -85,B 0,C 180,E1 24716.855,E2 24716.855} C_VEL
LIN {X 0,Y 542.232,Z 968.135,A -85,B 0,C 180,E1 24715.967,E2 24715.967} C_VEL
LIN {X 0,Y 558.266,Z 936.058,A -85,B 0,C 180,E1 24714.653,E2 24714.653} C_VEL
LIN {X 0,Y 562.932,Z 927.598,A -85,B 0,C 180,E1 24714.341,E2 24714.341} C_VEL
LIN {X 0,Y 553.837,Z 912.508,A -85,B 0,C 180,E1 24712.852,E2 24712.852} C_VEL
LIN {X 0,Y 546.481,Z 895.862,A -85,B 0,C 180,E1 24711.294,E2 24711.294} C_VEL
LIN {X 0,Y 541.14,Z 878.368,A -85,B 0,C 180,E1 24709.74,E2 24709.74} C_VEL
LIN {X 0,Y 537.535,Z 858.551,A -85,B 0,C 180,E1 24708.078,E2 24708.078} C_VEL
LIN {X 0,Y 536.086,Z 837.692,A -85,B 0,C 180,E1 24706.437,E2 24706.437} C_VEL
LIN {X 0,Y 536.674,Z 813.067,A -85,B 0,C 180,E1 24704.624,E2 24704.624} C_VEL
LIN {X 0,Y 543.378,Z 752.346,A -85,B 0,C 180,E1 24700.428,E2 24700.428} C_VEL
LIN {X 0,Y 543.217,Z 751.858,A -85,B 0,C 180,E1 24700.354,E2 24700.354} C_VEL
LIN {X 0,Y 544.897,Z 751.156,A -85,B 0,C 180,E1 24699.911,E2 24699.911} C_VEL
LIN {X 0,Y 546.78,Z 749.526,A -85,B 0,C 180,E1 24699.523,E2 24699.523} C_VEL
LIN {X 0,Y 549.614,Z 747.808,A -85,B 0,C 180,E1 24698.945,E2 24698.945} C_VEL
LIN {X 0,Y 552.088,Z 746.696,A -85,B 0,C 180,E1 24698.477,E2 24698.477} C_VEL
LIN {X 0,Y 553.108,Z 750.343,A -85,B 0,C 180,E1 24698.084,E2 24698.084} C_VEL
LIN {X 0,Y 553.111,Z 753.353,A -85,B 0,C 180,E1 24697.94,E2 24697.94} C_VEL
LIN {X 0,Y 543.356,Z 836.268,A -85,B 0,C 180,E1 24696.012,E2 24696.012} C_VEL
LIN {X 0,Y 536.275,Z 913.429,A -85,B 0,C 180,E1 24694.286,E2 24694.286} C_VEL
LIN {X 0,Y 531.1,Z 988.133,A -85,B 0,C 180,E1 24692.734,E2 24692.734} C_VEL
LIN {X 0,Y 529.017,Z 1022.901,A -85,B 0,C 180,E1 24691.993,E2 24691.993} C_VEL
LIN {X 0,Y 527.368,Z 1045.965,A -85,B 0,C 180,E1 24691.299,E2 24691.299} C_VEL
LIN {X 0,Y 525.376,Z 1068.462,A -85,B 0,C 180,E1 24690.414,E2 24690.414} C_VEL
LIN {X 0,Y 523.206,Z 1089.996,A -85,B 0,C 180,E1 24689.354,E2 24689.354} C_VEL
LIN {X 0,Y 520.882,Z 1110.639,A -85,B 0,C 180,E1 24688.117,E2 24688.117} C_VEL
LIN {X 0,Y 518.381,Z 1131.061,A -85,B 0,C 180,E1 24686.645,E2 24686.645} C_VEL
LIN {X 0,Y 515.97,Z 1149.644,A -85,B 0,C 180,E1 24685.051,E2 24685.051} C_VEL
LIN {X 0,Y 513.688,Z 1166.641,A -85,B 0,C 180,E1 24683.335,E2 24683.335} C_VEL
LIN {X 0,Y 511.506,Z 1182.517,A -85,B 0,C 180,E1 24681.441,E2 24681.441} C_VEL
LIN {X 0,Y 509.619,Z 1196.41,A -85,B 0,C 180,E1 24679.484,E2 24679.484} C_VEL
LIN {X 0,Y 507.912,Z 1209.579,A -85,B 0,C 180,E1 24677.293,E2 24677.293} C_VEL
LIN {X 0,Y 506.644,Z 1220.239,A -85,B 0,C 180,E1 24675.186,E2 24675.186} C_VEL
LIN {X 0,Y 505.625,Z 1229.751,A -85,B 0,C 180,E1 24672.912,E2 24672.912} C_VEL
LIN {X 0,Y 504.919,Z 1237.485,A -85,B 0,C 180,E1 24670.613,E2 24670.613} C_VEL
LIN {X 0,Y 504.456,Z 1243.818,A -85,B 0,C 180,E1 24668.205,E2 24668.205} C_VEL
LIN {X 0,Y 504.213,Z 1248.44,A -85,B 0,C 180,E1 24665.805,E2 24665.805} C_VEL
LIN {X 0,Y 504.078,Z 1251.288,A -85,B 0,C 180,E1 24663.412,E2 24663.412} C_VEL
LIN {X 0,Y 504.039,Z 1252.593,A -85,B 0,C 180,E1 24660.909,E2 24660.909} C_VEL
LIN {X 0,Y 504.025,Z 1252.328,A -85,B 0,C 180,E1 24658.636,E2 24658.636} C_VEL
LIN {X 0,Y 504.05,Z 1250.361,A -85,B 0,C 180,E1 24656.247,E2 24656.247} C_VEL
LIN {X 0,Y 504.146,Z 1246.818,A -85,B 0,C 180,E1 24653.852,E2 24653.852} C_VEL
LIN {X 0,Y 504.364,Z 1241.928,A -85,B 0,C 180,E1 24651.564,E2 24651.564} C_VEL
LIN {X 0,Y 504.744,Z 1235.291,A -85,B 0,C 180,E1 24649.268,E2 24649.268} C_VEL
